LIN {X 0.032,Y -299.569,Z 1828.357,A 0.000,B 0.000,C 90.000,E1 64.229} C_DIS
LIN {X -0.106,Y -287.457,Z 1828.340,A 0.000,B 0.000,C 90.000,E1 61.257} C_DIS
LIN {X -0.056,Y -278.078,Z 1828.327,A 0.000,B 0.000,C 90.000,E1 58.869} C_DIS
LIN {X 0.072,Y -268.639,Z 1828.313,A 0.000,B 0.000,C 90.000,E1 56.421} C_DIS
LIN {X 0.019,Y -260.469,Z 1828.302,A 0.000,B 0.000,C 90.000,E1 54.322} C_DIS
LIN {X -0.032,Y -252.251,Z 1828.290,A 0.000,B 0.000,C 90.000,E1 52.190} C_DIS
LIN {X -0.029,Y -249.462,Z 1828.286,A 0.000,B 0.000,C 90.000,E1 51.457} C_DIS
LIN {X -0.079,Y -249.453,Z 1828.286,A 0.000,B 0.000,C 90.000,E1 51.457} C_DIS
LIN {X 0.072,Y -254.487,Z 1828.280,A 0.000,B 0.000,C 90.000,E1 50.356} C_DIS
LIN {X -0.079,Y -255.818,Z 1828.276,A 0.000,B 0.000,C 90.000,E1 49.666} C_DIS
LIN {X -0.023,Y -255.690,Z 1828.272,A 0.000,B 0.000,C 90.000,E1 48.933} C_DIS
LIN {X -0.153,Y -255.059,Z 1828.268,A 0.000,B 0.000,C 90.000,E1 48.243} C_DIS
LIN {X 0.076,Y -254.151,Z 1828.264,A 0.000,B 0.000,C 90.000,E1 47.472} C_DIS
LIN {X -0.026,Y -251.829,Z 1828.256,A 0.000,B 0.000,C 90.000,E1 46.053} C_DIS
LIN {X 0.022,Y -249.143,Z 1828.248,A 0.000,B 0.000,C 90.000,E1 44.595} C_DIS
LIN {X 0.039,Y -244.690,Z 1828.236,A 0.000,B 0.000,C 90.000,E1 42.405} C_DIS
LIN {X -0.033,Y -239.918,Z 1828.223,A 0.000,B 0.000,C 90.000,E1 40.216} C_DIS
LIN {X -0.009,Y -233.391,Z 1828.207,A 0.000,B 0.000,C 90.000,E1 37.237} C_DIS
LIN {X 0.086,Y -226.660,Z 1828.190,A 0.000,B 0.000,C 90.000,E1 34.199} C_DIS
LIN {X 0.024,Y -221.773,Z 1828.177,A 0.000,B 0.000,C 90.000,E1 31.926} C_DIS
LIN {X 0.052,Y -213.666,Z 1828.156,A 0.000,B 0.000,C 90.000,E1 28.052} C_DIS
LIN {X 0.010,Y -206.205,Z 1828.134,A 0.000,B 0.000,C 90.000,E1 24.131} C_DIS
LIN {X 0.086,Y -200.971,Z 1828.116,A 0.000,B 0.000,C 90.000,E1 20.918} C_DIS
LIN {X -0.033,Y -195.411,Z 1828.094,A 0.000,B 0.000,C 90.000,E1 16.913} C_DIS
LIN {X -0.035,Y -191.019,Z 1828.071,A 0.000,B 0.000,C 90.000,E1 12.827} C_DIS
LIN {X 0.032,Y -187.518,Z 1828.048,A 0.000,B 0.000,C 90.000,E1 8.681} C_DIS
LIN {X -0.001,Y -184.293,Z 1828.016,A 0.000,B 0.000,C 90.000,E1 2.865} C_DIS
LIN {X 0.059,Y -182.919,Z 1827.979,A 0.000,B 0.000,C 90.000,E1 356.159} C_DIS
LIN {X -0.023,Y -183.519,Z 1827.937,A 0.000,B 0.000,C 90.000,E1 348.634} C_DIS
LIN {X -0.034,Y -184.958,Z 1827.909,A 0.000,B 0.000,C 90.000,E1 343.614} C_DIS
LIN {X 0.018,Y -187.227,Z 1827.881,A 0.000,B 0.000,C 90.000,E1 338.592} C_DIS
LIN {X -0.063,Y -190.361,Z 1827.853,A 0.000,B 0.000,C 90.000,E1 333.640} C_DIS
LIN {X 0.062,Y -194.276,Z 1827.826,A 0.000,B 0.000,C 90.000,E1 328.663} C_DIS
LIN {X -0.035,Y -198.125,Z 1827.803,A 0.000,B 0.000,C 90.000,E1 324.609} C_DIS
LIN {X -0.033,Y -202.723,Z 1827.781,A 0.000,B 0.000,C 90.000,E1 320.561} C_DIS
LIN {X 0.128,Y -207.396,Z 1827.763,A 0.000,B 0.000,C 90.000,E1 317.310} C_DIS
LIN {X 0.009,Y -211.919,Z 1827.750,A 0.000,B 0.000,C 90.000,E1 314.960} C_DIS
LIN {X -0.077,Y -216.582,Z 1827.739,A 0.000,B 0.000,C 90.000,E1 313.014} C_DIS
LIN {X 0.005,Y -221.156,Z 1827.730,A 0.000,B 0.000,C 90.000,E1 311.434} C_DIS
LIN {X 0.022,Y -226.545,Z 1827.722,A 0.000,B 0.000,C 90.000,E1 309.886} C_DIS
LIN {X -0.066,Y -232.712,Z 1827.713,A 0.000,B 0.000,C 90.000,E1 308.382} C_DIS
LIN {X 0.102,Y -243.179,Z 1827.701,A 0.000,B 0.000,C 90.000,E1 306.091} C_DIS
LIN {X -0.019,Y -252.825,Z 1827.690,A 0.000,B 0.000,C 90.000,E1 304.278} C_DIS
LIN {X -0.093,Y -265.541,Z 1827.678,A 0.000,B 0.000,C 90.000,E1 302.133} C_DIS
LIN {X -0.090,Y -284.139,Z 1827.663,A 0.000,B 0.000,C 90.000,E1 299.333} C_DIS
LIN {X 0.121,Y -298.703,Z 1827.652,A 0.000,B 0.000,C 90.000,E1 297.257} C_DIS
LIN {X -0.090,Y -311.079,Z 1827.642,A 0.000,B 0.000,C 90.000,E1 295.643} C_DIS
LIN {X -0.108,Y -323.475,Z 1827.633,A 0.000,B 0.000,C 90.000,E1 294.027} C_DIS
LIN {X 0.094,Y -335.710,Z 1827.625,A 0.000,B 0.000,C 90.000,E1 292.408} C_DIS
LIN {X 0.045,Y -345.213,Z 1827.618,A 0.000,B 0.000,C 90.000,E1 291.173} C_DIS
LIN {X 0.112,Y -354.151,Z 1827.611,A 0.000,B 0.000,C 90.000,E1 289.939} C_DIS
LIN {X 0.111,Y -360.270,Z 1827.606,A 0.000,B 0.000,C 90.000,E1 289.033} C_DIS
LIN {X -0.171,Y -365.811,Z 1827.601,A 0.000,B 0.000,C 90.000,E1 288.181} C_DIS
LIN {X -0.063,Y -370.611,Z 1827.596,A 0.000,B 0.000,C 90.000,E1 287.275} C_DIS
LIN {X -0.011,Y -374.520,Z 1827.591,A 0.000,B 0.000,C 90.000,E1 286.386} C_DIS
LIN {X 0.180,Y -377.576,Z 1827.586,A 0.000,B 0.000,C 90.000,E1 285.481} C_DIS
LIN {X -0.181,Y -379.206,Z 1827.583,A 0.000,B 0.000,C 90.000,E1 284.954} C_DIS
LIN {X -0.066,Y -380.464,Z 1827.580,A 0.000,B 0.000,C 90.000,E1 284.356} C_DIS
LIN {X -0.035,Y -381.302,Z 1827.577,A 0.000,B 0.000,C 90.000,E1 283.772} C_DIS
LIN {X 0.094,Y -381.711,Z 1827.573,A 0.000,B 0.000,C 90.000,E1 283.175} C_DIS
LIN {X 0.140,Y -381.680,Z 1827.570,A 0.000,B 0.000,C 90.000,E1 282.591} C_DIS
LIN {X -0.183,Y -381.269,Z 1827.567,A 0.000,B 0.000,C 90.000,E1 282.063} C_DIS
LIN {X -0.132,Y -380.387,Z 1827.564,A 0.000,B 0.000,C 90.000,E1 281.478} C_DIS
LIN {X -0.084,Y -379.051,Z 1827.560,A 0.000,B 0.000,C 90.000,E1 280.894} C_DIS
LIN {X -0.042,Y -377.252,Z 1827.557,A 0.000,B 0.000,C 90.000,E1 280.310} C_DIS
LIN {X -0.060,Y -373.979,Z 1827.552,A 0.000,B 0.000,C 90.000,E1 279.443} C_DIS
LIN {X -0.118,Y -367.706,Z 1827.544,A 0.000,B 0.000,C 90.000,E1 277.992} C_DIS
LIN {X 0.139,Y -363.441,Z 1827.539,A 0.000,B 0.000,C 90.000,E1 277.068} C_DIS
LIN {X 0.076,Y -360.186,Z 1827.536,A 0.000,B 0.000,C 90.000,E1 276.486} C_DIS
LIN {X -0.130,Y -354.419,Z 1827.531,A 0.000,B 0.000,C 90.000,E1 275.625} C_DIS
LIN {X 0.069,Y -349.826,Z 1827.528,A 0.000,B 0.000,C 90.000,E1 274.992} C_DIS
LIN {X -0.106,Y -344.534,Z 1827.524,A 0.000,B 0.000,C 90.000,E1 274.416} C_DIS
LIN {X 0.153,Y -338.687,Z 1827.521,A 0.000,B 0.000,C 90.000,E1 273.784} C_DIS
LIN {X 0.006,Y -332.711,Z 1827.518,A 0.000,B 0.000,C 90.000,E1 273.269} C_DIS
LIN {X 0.134,Y -326.424,Z 1827.515,A 0.000,B 0.000,C 90.000,E1 272.751} C_DIS
LIN {X -0.129,Y -319.978,Z 1827.513,A 0.000,B 0.000,C 90.000,E1 272.350} C_DIS
LIN {X -0.138,Y -313.290,Z 1827.511,A 0.000,B 0.000,C 90.000,E1 271.949} C_DIS
LIN {X 0.132,Y -306.164,Z 1827.509,A 0.000,B 0.000,C 90.000,E1 271.547} C_DIS
LIN {X 0.043,Y -298.467,Z 1827.507,A 0.000,B 0.000,C 90.000,E1 271.260} C_DIS
LIN {X 0.041,Y -291.054,Z 1827.506,A 0.000,B 0.000,C 90.000,E1 271.031} C_DIS
LIN {X 0.116,Y -279.908,Z 1827.504,A 0.000,B 0.000,C 90.000,E1 270.745} C_DIS
LIN {X -0.065,Y -250.463,Z 1827.501,A 0.000,B 0.000,C 90.000,E1 270.229} C_DIS
LIN {X -0.110,Y -240.845,Z 1827.500,A 0.000,B 0.000,C 90.000,E1 270.115} C_DIS
LIN {X -0.045,Y -234.411,Z 1827.500,A 0.000,B 0.000,C 90.000,E1 270.057} C_DIS
LIN {X -0.062,Y -181.566,Z 1827.500,A 0.000,B 0.000,C 90.000,E1 270.057} C_DIS
LIN {X 0.021,Y -180.907,Z 1827.475,A 0.000,B 0.000,C 90.000,E1 265.469} C_DIS
LIN {X 0.079,Y -180.739,Z 1827.470,A 0.000,B 0.000,C 90.000,E1 264.609} C_DIS
LIN {X 0.000,Y -178.830,Z 1827.442,A 0.000,B 0.000,C 90.000,E1 259.567} C_DIS
LIN {X 0.033,Y -175.874,Z 1827.414,A 0.000,B 0.000,C 90.000,E1 254.464} C_DIS
LIN {X -0.090,Y -173.848,Z 1827.400,A 0.000,B 0.000,C 90.000,E1 251.945} C_DIS
LIN {X 0.064,Y -171.516,Z 1827.380,A 0.000,B 0.000,C 90.000,E1 248.465} C_DIS
LIN {X 0.049,Y -167.743,Z 1827.356,A 0.000,B 0.000,C 90.000,E1 244.152} C_DIS
LIN {X 0.065,Y -166.444,Z 1827.347,A 0.000,B 0.000,C 90.000,E1 242.410} C_DIS
LIN {X -0.021,Y -163.161,Z 1827.327,A 0.000,B 0.000,C 90.000,E1 238.948} C_DIS
LIN {X 0.028,Y -161.119,Z 1827.313,A 0.000,B 0.000,C 90.000,E1 236.294} C_DIS
LIN {X -0.069,Y -157.143,Z 1827.288,A 0.000,B 0.000,C 90.000,E1 231.904} C_DIS
LIN {X -0.046,Y -155.876,Z 1827.278,A 0.000,B 0.000,C 90.000,E1 230.114} C_DIS
LIN {X -0.087,Y -152.125,Z 1827.253,A 0.000,B 0.000,C 90.000,E1 225.648} C_DIS
LIN {X -0.067,Y -150.375,Z 1827.238,A 0.000,B 0.000,C 90.000,E1 222.933} C_DIS
LIN {X -0.042,Y -147.109,Z 1827.213,A 0.000,B 0.000,C 90.000,E1 218.382} C_DIS
LIN {X 0.068,Y -145.676,Z 1827.198,A 0.000,B 0.000,C 90.000,E1 215.598} C_DIS
LIN {X -0.052,Y -143.058,Z 1827.172,A 0.000,B 0.000,C 90.000,E1 211.052} C_DIS
LIN {X 0.006,Y -141.680,Z 1827.152,A 0.000,B 0.000,C 90.000,E1 207.334} C_DIS
LIN {X -0.016,Y -139.457,Z 1827.116,A 0.000,B 0.000,C 90.000,E1 200.844} C_DIS
LIN {X 0.035,Y -139.190,Z 1827.105,A 0.000,B 0.000,C 90.000,E1 198.960} C_DIS
LIN {X 0.058,Y -138.324,Z 1827.054,A 0.000,B 0.000,C 90.000,E1 189.613} C_DIS
LIN {X 0.066,Y -139.456,Z 1827.007,A 0.000,B 0.000,C 90.000,E1 181.203} C_DIS
LIN {X 0.007,Y -141.006,Z 1826.976,A 0.000,B 0.000,C 90.000,E1 175.641} C_DIS
LIN {X -0.044,Y -142.760,Z 1826.955,A 0.000,B 0.000,C 90.000,E1 171.951} C_DIS
LIN {X 0.053,Y -145.165,Z 1826.930,A 0.000,B 0.000,C 90.000,E1 167.297} C_DIS
LIN {X 0.045,Y -147.787,Z 1826.909,A 0.000,B 0.000,C 90.000,E1 163.630} C_DIS
LIN {X -0.018,Y -150.468,Z 1826.889,A 0.000,B 0.000,C 90.000,E1 160.007} C_DIS
LIN {X 0.056,Y -153.921,Z 1826.869,A 0.000,B 0.000,C 90.000,E1 156.357} C_DIS
LIN {X -0.020,Y -157.331,Z 1826.849,A 0.000,B 0.000,C 90.000,E1 152.794} C_DIS
LIN {X 0.065,Y -161.522,Z 1826.829,A 0.000,B 0.000,C 90.000,E1 149.203} C_DIS
LIN {X 0.078,Y -165.721,Z 1826.809,A 0.000,B 0.000,C 90.000,E1 145.674} C_DIS
LIN {X 0.066,Y -170.669,Z 1826.790,A 0.000,B 0.000,C 90.000,E1 142.190} C_DIS
LIN {X -0.021,Y -175.544,Z 1826.771,A 0.000,B 0.000,C 90.000,E1 138.771} C_DIS
LIN {X 0.099,Y -181.163,Z 1826.752,A 0.000,B 0.000,C 90.000,E1 135.324} C_DIS
LIN {X -0.031,Y -186.618,Z 1826.733,A 0.000,B 0.000,C 90.000,E1 132.000} C_DIS
LIN {X 0.039,Y -191.227,Z 1826.719,A 0.000,B 0.000,C 90.000,E1 129.483} C_DIS
LIN {X -0.039,Y -197.042,Z 1826.701,A 0.000,B 0.000,C 90.000,E1 126.217} C_DIS
LIN {X -0.121,Y -200.314,Z 1826.692,A 0.000,B 0.000,C 90.000,E1 124.612} C_DIS
LIN {X 0.050,Y -207.804,Z 1826.670,A 0.000,B 0.000,C 90.000,E1 120.541} C_DIS
LIN {X 0.057,Y -210.971,Z 1826.661,A 0.000,B 0.000,C 90.000,E1 118.949} C_DIS
LIN {X 0.072,Y -216.849,Z 1826.643,A 0.000,B 0.000,C 90.000,E1 115.796} C_DIS
LIN {X 0.026,Y -218.465,Z 1826.639,A 0.000,B 0.000,C 90.000,E1 115.027} C_DIS
LIN {X 0.067,Y -221.183,Z 1826.630,A 0.000,B 0.000,C 90.000,E1 113.462} C_DIS
LIN {X -0.050,Y -224.036,Z 1826.622,A 0.000,B 0.000,C 90.000,E1 111.897} C_DIS
LIN {X -0.098,Y -283.686,Z 1826.622,A 0.000,B 0.000,C 90.000,E1 111.897} C_DIS
LIN {X 0.024,Y -285.203,Z 1826.621,A 0.000,B 0.000,C 90.000,E1 111.844} C_DIS
LIN {X 0.074,Y -288.957,Z 1826.620,A 0.000,B 0.000,C 90.000,E1 111.663} C_DIS
LIN {X -0.144,Y -291.142,Z 1826.620,A 0.000,B 0.000,C 90.000,E1 111.535} C_DIS
LIN {X 0.064,Y -294.171,Z 1826.618,A 0.000,B 0.000,C 90.000,E1 111.153} C_DIS
LIN {X 0.041,Y -296.176,Z 1826.616,A 0.000,B 0.000,C 90.000,E1 110.844} C_DIS
LIN {X 0.051,Y -309.270,Z 1826.603,A 0.000,B 0.000,C 90.000,E1 108.544} C_DIS
LIN {X 0.157,Y -323.836,Z 1826.590,A 0.000,B 0.000,C 90.000,E1 106.260} C_DIS
LIN {X -0.113,Y -337.506,Z 1826.580,A 0.000,B 0.000,C 90.000,E1 104.411} C_DIS
LIN {X 0.033,Y -352.360,Z 1826.570,A 0.000,B 0.000,C 90.000,E1 102.535} C_DIS
LIN {X 0.042,Y -370.762,Z 1826.558,A 0.000,B 0.000,C 90.000,E1 100.489} C_DIS
LIN {X 0.113,Y -389.583,Z 1826.548,A 0.000,B 0.000,C 90.000,E1 98.624} C_DIS
LIN {X 0.008,Y -408.823,Z 1826.539,A 0.000,B 0.000,C 90.000,E1 96.947} C_DIS
LIN {X -0.185,Y -431.190,Z 1826.529,A 0.000,B 0.000,C 90.000,E1 95.220} C_DIS
LIN {X -0.025,Y -439.544,Z 1826.526,A 0.000,B 0.000,C 90.000,E1 94.588} C_DIS
LIN {X 0.191,Y -441.622,Z 1826.524,A 0.000,B 0.000,C 90.000,E1 94.359} C_DIS
LIN {X 0.043,Y -443.572,Z 1826.523,A 0.000,B 0.000,C 90.000,E1 94.131} C_DIS
LIN {X -0.076,Y -445.062,Z 1826.522,A 0.000,B 0.000,C 90.000,E1 93.898} C_DIS
LIN {X 0.104,Y -446.265,Z 1826.520,A 0.000,B 0.000,C 90.000,E1 93.612} C_DIS
LIN {X -0.161,Y -447.151,Z 1826.519,A 0.000,B 0.000,C 90.000,E1 93.383} C_DIS
LIN {X -0.205,Y -448.124,Z 1826.516,A 0.000,B 0.000,C 90.000,E1 92.865} C_DIS
LIN {X 0.183,Y -448.151,Z 1826.513,A 0.000,B 0.000,C 90.000,E1 92.293} C_DIS
LIN {X 0.144,Y -447.239,Z 1826.510,A 0.000,B 0.000,C 90.000,E1 91.776} C_DIS
LIN {X 0.091,Y -445.244,Z 1826.507,A 0.000,B 0.000,C 90.000,E1 91.260} C_DIS
LIN {X -0.041,Y -438.759,Z 1826.501,A 0.000,B 0.000,C 90.000,E1 90.229} C_DIS
LIN {X 0.192,Y -427.223,Z 1826.491,A 0.000,B 0.000,C 90.000,E1 88.339} C_DIS
LIN {X -0.201,Y -415.449,Z 1826.480,A 0.000,B 0.000,C 90.000,E1 86.502} C_DIS
LIN {X 0.029,Y -403.593,Z 1826.470,A 0.000,B 0.000,C 90.000,E1 84.546} C_DIS
LIN {X 0.006,Y -391.662,Z 1826.459,A 0.000,B 0.000,C 90.000,E1 82.591} C_DIS
LIN {X -0.174,Y -379.704,Z 1826.448,A 0.000,B 0.000,C 90.000,E1 80.622} C_DIS
LIN {X -0.113,Y -364.559,Z 1826.433,A 0.000,B 0.000,C 90.000,E1 77.993} C_DIS
LIN {X 0.006,Y -347.149,Z 1826.415,A 0.000,B 0.000,C 90.000,E1 74.685} C_DIS
LIN {X -0.011,Y -335.109,Z 1826.401,A 0.000,B 0.000,C 90.000,E1 72.236} C_DIS
LIN {X -0.116,Y -323.322,Z 1826.387,A 0.000,B 0.000,C 90.000,E1 69.752} C_DIS
LIN {X -0.027,Y -309.201,Z 1826.370,A 0.000,B 0.000,C 90.000,E1 66.538} C_DIS
LIN {X -0.176,Y -299.597,Z 1826.357,A 0.000,B 0.000,C 90.000,E1 64.280} C_DIS
LIN {X -0.044,Y -287.482,Z 1826.340,A 0.000,B 0.000,C 90.000,E1 61.257} C_DIS
LIN {X 0.004,Y -278.105,Z 1826.327,A 0.000,B 0.000,C 90.000,E1 58.869} C_DIS
LIN {X 0.130,Y -268.669,Z 1826.314,A 0.000,B 0.000,C 90.000,E1 56.421} C_DIS
LIN {X 0.077,Y -260.499,Z 1826.302,A 0.000,B 0.000,C 90.000,E1 54.322} C_DIS
LIN {X 0.062,Y -256.702,Z 1826.296,A 0.000,B 0.000,C 90.000,E1 53.336} C_DIS
LIN {X 0.012,Y -256.683,Z 1826.296,A 0.000,B 0.000,C 90.000,E1 53.336} C_DIS
LIN {X 0.030,Y -261.851,Z 1826.290,A 0.000,B 0.000,C 90.000,E1 52.190} C_DIS
LIN {X 0.074,Y -262.675,Z 1826.288,A 0.000,B 0.000,C 90.000,E1 51.823} C_DIS
LIN {X 0.015,Y -262.863,Z 1826.284,A 0.000,B 0.000,C 90.000,E1 51.126} C_DIS
LIN {X -0.079,Y -262.317,Z 1826.280,A 0.000,B 0.000,C 90.000,E1 50.436} C_DIS
LIN {X 0.032,Y -261.416,Z 1826.276,A 0.000,B 0.000,C 90.000,E1 49.703} C_DIS
LIN {X -0.158,Y -259.054,Z 1826.268,A 0.000,B 0.000,C 90.000,E1 48.324} C_DIS
LIN {X -0.009,Y -256.276,Z 1826.260,A 0.000,B 0.000,C 90.000,E1 46.863} C_DIS
LIN {X 0.133,Y -251.648,Z 1826.248,A 0.000,B 0.000,C 90.000,E1 44.676} C_DIS
LIN {X 0.012,Y -246.729,Z 1826.236,A 0.000,B 0.000,C 90.000,E1 42.528} C_DIS
LIN {X 0.002,Y -241.617,Z 1826.224,A 0.000,B 0.000,C 90.000,E1 40.334} C_DIS
LIN {X 0.032,Y -234.705,Z 1826.208,A 0.000,B 0.000,C 90.000,E1 37.363} C_DIS
LIN {X 0.025,Y -227.628,Z 1826.191,A 0.000,B 0.000,C 90.000,E1 34.358} C_DIS
LIN {X -0.014,Y -222.517,Z 1826.178,A 0.000,B 0.000,C 90.000,E1 32.084} C_DIS
LIN {X -0.042,Y -214.038,Z 1826.157,A 0.000,B 0.000,C 90.000,E1 28.231} C_DIS
LIN {X 0.026,Y -206.204,Z 1826.135,A 0.000,B 0.000,C 90.000,E1 24.283} C_DIS
LIN {X -0.002,Y -200.772,Z 1826.117,A 0.000,B 0.000,C 90.000,E1 21.099} C_DIS
LIN {X 0.062,Y -195.153,Z 1826.095,A 0.000,B 0.000,C 90.000,E1 17.040} C_DIS
LIN {X 0.056,Y -190.746,Z 1826.072,A 0.000,B 0.000,C 90.000,E1 12.952} C_DIS
LIN {X -0.064,Y -187.228,Z 1826.049,A 0.000,B 0.000,C 90.000,E1 8.859} C_DIS
LIN {X -0.087,Y -183.950,Z 1826.017,A 0.000,B 0.000,C 90.000,E1 3.037} C_DIS
LIN {X 0.049,Y -182.523,Z 1825.979,A 0.000,B 0.000,C 90.000,E1 356.159} C_DIS
LIN {X -0.054,Y -183.146,Z 1825.937,A 0.000,B 0.000,C 90.000,E1 348.634} C_DIS
LIN {X 0.097,Y -184.598,Z 1825.909,A 0.000,B 0.000,C 90.000,E1 343.559} C_DIS
LIN {X -0.041,Y -186.900,Z 1825.881,A 0.000,B 0.000,C 90.000,E1 338.592} C_DIS
LIN {X 0.035,Y -190.071,Z 1825.853,A 0.000,B 0.000,C 90.000,E1 333.589} C_DIS
LIN {X -0.023,Y -194.016,Z 1825.826,A 0.000,B 0.000,C 90.000,E1 328.663} C_DIS
LIN {X 0.032,Y -197.887,Z 1825.803,A 0.000,B 0.000,C 90.000,E1 324.562} C_DIS
LIN {X 0.021,Y -202.562,Z 1825.781,A 0.000,B 0.000,C 90.000,E1 320.517} C_DIS
LIN {X 0.019,Y -207.333,Z 1825.763,A 0.000,B 0.000,C 90.000,E1 317.310} C_DIS
LIN {X 0.047,Y -211.950,Z 1825.750,A 0.000,B 0.000,C 90.000,E1 314.919} C_DIS
LIN {X -0.043,Y -216.696,Z 1825.739,A 0.000,B 0.000,C 90.000,E1 312.975} C_DIS
LIN {X 0.055,Y -221.326,Z 1825.730,A 0.000,B 0.000,C 90.000,E1 311.391} C_DIS
LIN {X 0.052,Y -226.748,Z 1825.721,A 0.000,B 0.000,C 90.000,E1 309.850} C_DIS
LIN {X 0.001,Y -232.962,Z 1825.713,A 0.000,B 0.000,C 90.000,E1 308.338} C_DIS
LIN {X -0.015,Y -243.483,Z 1825.700,A 0.000,B 0.000,C 90.000,E1 306.091} C_DIS
LIN {X 0.007,Y -253.163,Z 1825.690,A 0.000,B 0.000,C 90.000,E1 304.246} C_DIS
LIN {X 0.122,Y -263.710,Z 1825.680,A 0.000,B 0.000,C 90.000,E1 302.418} C_DIS
LIN {X -0.147,Y -282.183,Z 1825.665,A 0.000,B 0.000,C 90.000,E1 299.667} C_DIS
LIN {X 0.024,Y -296.726,Z 1825.653,A 0.000,B 0.000,C 90.000,E1 297.590} C_DIS
LIN {X 0.084,Y -311.609,Z 1825.642,A 0.000,B 0.000,C 90.000,E1 295.591} C_DIS
LIN {X -0.079,Y -324.054,Z 1825.633,A 0.000,B 0.000,C 90.000,E1 294.003} C_DIS
LIN {X -0.002,Y -336.339,Z 1825.625,A 0.000,B 0.000,C 90.000,E1 292.408} C_DIS
LIN {X 0.079,Y -345.855,Z 1825.618,A 0.000,B 0.000,C 90.000,E1 291.153} C_DIS
LIN {X -0.006,Y -352.657,Z 1825.612,A 0.000,B 0.000,C 90.000,E1 290.248} C_DIS
LIN {X 0.104,Y -358.959,Z 1825.607,A 0.000,B 0.000,C 90.000,E1 289.322} C_DIS
LIN {X 0.146,Y -364.726,Z 1825.602,A 0.000,B 0.000,C 90.000,E1 288.417} C_DIS
LIN {X 0.171,Y -368.168,Z 1825.599,A 0.000,B 0.000,C 90.000,E1 287.819} C_DIS
LIN {X -0.134,Y -371.253,Z 1825.596,A 0.000,B 0.000,C 90.000,E1 287.275} C_DIS
LIN {X -0.068,Y -373.930,Z 1825.593,A 0.000,B 0.000,C 90.000,E1 286.677} C_DIS
LIN {X 0.019,Y -376.221,Z 1825.589,A 0.000,B 0.000,C 90.000,E1 286.079} C_DIS
LIN {X 0.119,Y -378.160,Z 1825.586,A 0.000,B 0.000,C 90.000,E1 285.481} C_DIS
LIN {X 0.128,Y -379.776,Z 1825.583,A 0.000,B 0.000,C 90.000,E1 284.898} C_DIS
LIN {X -0.121,Y -381.028,Z 1825.580,A 0.000,B 0.000,C 90.000,E1 284.356} C_DIS
LIN {X -0.087,Y -381.860,Z 1825.576,A 0.000,B 0.000,C 90.000,E1 283.772} C_DIS
LIN {X 0.046,Y -382.226,Z 1825.573,A 0.000,B 0.000,C 90.000,E1 283.175} C_DIS
LIN {X 0.096,Y -382.215,Z 1825.570,A 0.000,B 0.000,C 90.000,E1 282.591} C_DIS
LIN {X 0.149,Y -381.750,Z 1825.567,A 0.000,B 0.000,C 90.000,E1 282.007} C_DIS
LIN {X -0.170,Y -380.851,Z 1825.564,A 0.000,B 0.000,C 90.000,E1 281.478} C_DIS
LIN {X -0.119,Y -379.489,Z 1825.560,A 0.000,B 0.000,C 90.000,E1 280.894} C_DIS
LIN {X -0.074,Y -377.763,Z 1825.557,A 0.000,B 0.000,C 90.000,E1 280.310} C_DIS
LIN {X -0.088,Y -374.470,Z 1825.552,A 0.000,B 0.000,C 90.000,E1 279.443} C_DIS
LIN {X -0.137,Y -368.145,Z 1825.544,A 0.000,B 0.000,C 90.000,E1 277.992} C_DIS
LIN {X 0.124,Y -363.786,Z 1825.539,A 0.000,B 0.000,C 90.000,E1 277.068} C_DIS
LIN {X -0.013,Y -358.692,Z 1825.534,A 0.000,B 0.000,C 90.000,E1 276.201} C_DIS
LIN {X -0.140,Y -354.694,Z 1825.531,A 0.000,B 0.000,C 90.000,E1 275.625} C_DIS
LIN {X 0.062,Y -350.026,Z 1825.528,A 0.000,B 0.000,C 90.000,E1 274.992} C_DIS
LIN {X -0.014,Y -344.864,Z 1825.525,A 0.000,B 0.000,C 90.000,E1 274.416} C_DIS
LIN {X -0.067,Y -339.090,Z 1825.521,A 0.000,B 0.000,C 90.000,E1 273.841} C_DIS
LIN {X 0.095,Y -333.057,Z 1825.518,A 0.000,B 0.000,C 90.000,E1 273.269} C_DIS
LIN {X -0.101,Y -326.828,Z 1825.516,A 0.000,B 0.000,C 90.000,E1 272.808} C_DIS
LIN {X -0.058,Y -320.291,Z 1825.513,A 0.000,B 0.000,C 90.000,E1 272.350} C_DIS
LIN {X -0.029,Y -313.795,Z 1825.511,A 0.000,B 0.000,C 90.000,E1 271.949} C_DIS
LIN {X -0.081,Y -306.654,Z 1825.509,A 0.000,B 0.000,C 90.000,E1 271.604} C_DIS
LIN {X -0.133,Y -299.165,Z 1825.507,A 0.000,B 0.000,C 90.000,E1 271.318} C_DIS
LIN {X 0.139,Y -291.851,Z 1825.506,A 0.000,B 0.000,C 90.000,E1 271.031} C_DIS
LIN {X -0.083,Y -280.769,Z 1825.504,A 0.000,B 0.000,C 90.000,E1 270.802} C_DIS
LIN {X 0.009,Y -251.290,Z 1825.501,A 0.000,B 0.000,C 90.000,E1 270.229} C_DIS
LIN {X -0.042,Y -241.853,Z 1825.501,A 0.000,B 0.000,C 90.000,E1 270.115} C_DIS
LIN {X -0.019,Y -233.753,Z 1825.500,A 0.000,B 0.000,C 90.000,E1 270.057} C_DIS
LIN {X -0.042,Y -181.567,Z 1825.500,A 0.000,B 0.000,C 90.000,E1 270.057} C_DIS
LIN {X 0.066,Y -180.907,Z 1825.475,A 0.000,B 0.000,C 90.000,E1 265.469} C_DIS
LIN {X -0.056,Y -180.746,Z 1825.470,A 0.000,B 0.000,C 90.000,E1 264.666} C_DIS
LIN {X 0.012,Y -178.837,Z 1825.442,A 0.000,B 0.000,C 90.000,E1 259.577} C_DIS
LIN {X -0.092,Y -175.881,Z 1825.414,A 0.000,B 0.000,C 90.000,E1 254.519} C_DIS
LIN {X 0.015,Y -174.544,Z 1825.404,A 0.000,B 0.000,C 90.000,E1 252.779} C_DIS
LIN {X -0.053,Y -171.528,Z 1825.381,A 0.000,B 0.000,C 90.000,E1 248.518} C_DIS
LIN {X -0.059,Y -167.753,Z 1825.357,A 0.000,B 0.000,C 90.000,E1 244.204} C_DIS
LIN {X 0.031,Y -166.458,Z 1825.347,A 0.000,B 0.000,C 90.000,E1 242.436} C_DIS
LIN {X 0.021,Y -163.173,Z 1825.328,A 0.000,B 0.000,C 90.000,E1 238.948} C_DIS
LIN {X 0.070,Y -161.133,Z 1825.313,A 0.000,B 0.000,C 90.000,E1 236.294} C_DIS
LIN {X -0.027,Y -157.154,Z 1825.288,A 0.000,B 0.000,C 90.000,E1 231.904} C_DIS
LIN {X -0.004,Y -155.887,Z 1825.278,A 0.000,B 0.000,C 90.000,E1 230.114} C_DIS
LIN {X -0.046,Y -152.137,Z 1825.254,A 0.000,B 0.000,C 90.000,E1 225.648} C_DIS
LIN {X -0.026,Y -150.386,Z 1825.238,A 0.000,B 0.000,C 90.000,E1 222.933} C_DIS
LIN {X -0.002,Y -147.117,Z 1825.213,A 0.000,B 0.000,C 90.000,E1 218.382} C_DIS
LIN {X -0.011,Y -145.683,Z 1825.198,A 0.000,B 0.000,C 90.000,E1 215.644} C_DIS
LIN {X -0.012,Y -143.065,Z 1825.172,A 0.000,B 0.000,C 90.000,E1 211.052} C_DIS
LIN {X 0.045,Y -141.687,Z 1825.152,A 0.000,B 0.000,C 90.000,E1 207.334} C_DIS
LIN {X -0.027,Y -139.460,Z 1825.116,A 0.000,B 0.000,C 90.000,E1 200.865} C_DIS
LIN {X 0.074,Y -139.193,Z 1825.105,A 0.000,B 0.000,C 90.000,E1 198.960} C_DIS
LIN {X -0.040,Y -138.324,Z 1825.054,A 0.000,B 0.000,C 90.000,E1 189.670} C_DIS
LIN {X -0.035,Y -139.453,Z 1825.007,A 0.000,B 0.000,C 90.000,E1 181.260} C_DIS
LIN {X 0.045,Y -140.999,Z 1824.976,A 0.000,B 0.000,C 90.000,E1 175.641} C_DIS
LIN {X -0.005,Y -142.754,Z 1824.955,A 0.000,B 0.000,C 90.000,E1 171.951} C_DIS
LIN {X -0.050,Y -145.156,Z 1824.930,A 0.000,B 0.000,C 90.000,E1 167.353} C_DIS
LIN {X -0.056,Y -147.778,Z 1824.909,A 0.000,B 0.000,C 90.000,E1 163.685} C_DIS
LIN {X 0.023,Y -150.455,Z 1824.889,A 0.000,B 0.000,C 90.000,E1 160.007} C_DIS
LIN {X -0.044,Y -153.905,Z 1824.869,A 0.000,B 0.000,C 90.000,E1 156.410} C_DIS
LIN {X 0.022,Y -157.315,Z 1824.849,A 0.000,B 0.000,C 90.000,E1 152.794} C_DIS
LIN {X -0.032,Y -161.502,Z 1824.829,A 0.000,B 0.000,C 90.000,E1 149.253} C_DIS
LIN {X -0.017,Y -165.702,Z 1824.810,A 0.000,B 0.000,C 90.000,E1 145.722} C_DIS
LIN {X 0.110,Y -170.646,Z 1824.790,A 0.000,B 0.000,C 90.000,E1 142.190} C_DIS
LIN {X 0.023,Y -175.522,Z 1824.771,A 0.000,B 0.000,C 90.000,E1 138.771} C_DIS
LIN {X 0.017,Y -181.142,Z 1824.752,A 0.000,B 0.000,C 90.000,E1 135.364} C_DIS
LIN {X 0.015,Y -186.593,Z 1824.733,A 0.000,B 0.000,C 90.000,E1 132.000} C_DIS
LIN {X 0.085,Y -191.204,Z 1824.719,A 0.000,B 0.000,C 90.000,E1 129.483} C_DIS
LIN {X 0.009,Y -197.015,Z 1824.701,A 0.000,B 0.000,C 90.000,E1 126.217} C_DIS
LIN {X -0.073,Y -200.285,Z 1824.692,A 0.000,B 0.000,C 90.000,E1 124.612} C_DIS
LIN {X -0.080,Y -207.776,Z 1824.670,A 0.000,B 0.000,C 90.000,E1 120.590} C_DIS
LIN {X 0.106,Y -210.948,Z 1824.661,A 0.000,B 0.000,C 90.000,E1 118.949} C_DIS
LIN {X -0.073,Y -216.822,Z 1824.643,A 0.000,B 0.000,C 90.000,E1 115.848} C_DIS
LIN {X 0.075,Y -218.437,Z 1824.639,A 0.000,B 0.000,C 90.000,E1 115.027} C_DIS
LIN {X -0.085,Y -221.160,Z 1824.630,A 0.000,B 0.000,C 90.000,E1 113.515} C_DIS
LIN {X -0.027,Y -224.024,Z 1824.622,A 0.000,B 0.000,C 90.000,E1 111.897} C_DIS
LIN {X -0.069,Y -283.207,Z 1824.622,A 0.000,B 0.000,C 90.000,E1 111.897} C_DIS
LIN {X 0.089,Y -284.723,Z 1824.621,A 0.000,B 0.000,C 90.000,E1 111.844} C_DIS
LIN {X -0.128,Y -288.773,Z 1824.620,A 0.000,B 0.000,C 90.000,E1 111.716} C_DIS
LIN {X -0.078,Y -291.007,Z 1824.620,A 0.000,B 0.000,C 90.000,E1 111.535} C_DIS
LIN {X 0.024,Y -294.077,Z 1824.618,A 0.000,B 0.000,C 90.000,E1 111.173} C_DIS
LIN {X 0.019,Y -296.084,Z 1824.616,A 0.000,B 0.000,C 90.000,E1 110.865} C_DIS
LIN {X 0.153,Y -309.155,Z 1824.603,A 0.000,B 0.000,C 90.000,E1 108.544} C_DIS
LIN {X -0.049,Y -323.709,Z 1824.591,A 0.000,B 0.000,C 90.000,E1 106.315} C_DIS
LIN {X -0.006,Y -337.368,Z 1824.580,A 0.000,B 0.000,C 90.000,E1 104.411} C_DIS
LIN {X 0.141,Y -352.210,Z 1824.570,A 0.000,B 0.000,C 90.000,E1 102.535} C_DIS
LIN {X 0.146,Y -370.606,Z 1824.558,A 0.000,B 0.000,C 90.000,E1 100.489} C_DIS
LIN {X 0.213,Y -389.424,Z 1824.548,A 0.000,B 0.000,C 90.000,E1 98.624} C_DIS
LIN {X 0.103,Y -408.661,Z 1824.539,A 0.000,B 0.000,C 90.000,E1 96.947} C_DIS
LIN {X -0.094,Y -431.025,Z 1824.529,A 0.000,B 0.000,C 90.000,E1 95.220} C_DIS
LIN {X 0.063,Y -439.402,Z 1824.526,A 0.000,B 0.000,C 90.000,E1 94.588} C_DIS
LIN {X -0.162,Y -441.511,Z 1824.524,A 0.000,B 0.000,C 90.000,E1 94.416} C_DIS
LIN {X 0.149,Y -443.470,Z 1824.523,A 0.000,B 0.000,C 90.000,E1 94.131} C_DIS
LIN {X 0.049,Y -444.968,Z 1824.522,A 0.000,B 0.000,C 90.000,E1 93.898} C_DIS
LIN {X -0.216,Y -446.191,Z 1824.520,A 0.000,B 0.000,C 90.000,E1 93.669} C_DIS
LIN {X -0.036,Y -447.094,Z 1824.519,A 0.000,B 0.000,C 90.000,E1 93.383} C_DIS
LIN {X -0.079,Y -448.096,Z 1824.516,A 0.000,B 0.000,C 90.000,E1 92.865} C_DIS
LIN {X -0.140,Y -448.149,Z 1824.513,A 0.000,B 0.000,C 90.000,E1 92.350} C_DIS
LIN {X -0.178,Y -447.266,Z 1824.510,A 0.000,B 0.000,C 90.000,E1 91.833} C_DIS
LIN {X 0.215,Y -445.306,Z 1824.507,A 0.000,B 0.000,C 90.000,E1 91.260} C_DIS
LIN {X -0.101,Y -440.496,Z 1824.503,A 0.000,B 0.000,C 90.000,E1 90.516} C_DIS
LIN {X 0.176,Y -428.964,Z 1824.492,A 0.000,B 0.000,C 90.000,E1 88.625} C_DIS
LIN {X -0.188,Y -417.204,Z 1824.482,A 0.000,B 0.000,C 90.000,E1 86.788} C_DIS
LIN {X -0.016,Y -407.075,Z 1824.473,A 0.000,B 0.000,C 90.000,E1 85.122} C_DIS
LIN {X 0.038,Y -395.163,Z 1824.462,A 0.000,B 0.000,C 90.000,E1 83.166} C_DIS
LIN {X -0.068,Y -383.207,Z 1824.451,A 0.000,B 0.000,C 90.000,E1 81.197} C_DIS
LIN {X 0.023,Y -369.613,Z 1824.438,A 0.000,B 0.000,C 90.000,E1 78.870} C_DIS
LIN {X 0.132,Y -351.845,Z 1824.420,A 0.000,B 0.000,C 90.000,E1 75.589} C_DIS
LIN {X 0.109,Y -338.160,Z 1824.405,A 0.000,B 0.000,C 90.000,E1 72.851} C_DIS
LIN {X 0.099,Y -327.784,Z 1824.393,A 0.000,B 0.000,C 90.000,E1 70.678} C_DIS
LIN {X -0.102,Y -313.419,Z 1824.375,A 0.000,B 0.000,C 90.000,E1 67.539} C_DIS
LIN {X 0.013,Y -302.403,Z 1824.361,A 0.000,B 0.000,C 90.000,E1 64.921} C_DIS
LIN {X -0.042,Y -290.191,Z 1824.344,A 0.000,B 0.000,C 90.000,E1 61.948} C_DIS
LIN {X -0.066,Y -280.836,Z 1824.331,A 0.000,B 0.000,C 90.000,E1 59.587} C_DIS
LIN {X -0.017,Y -271.430,Z 1824.318,A 0.000,B 0.000,C 90.000,E1 57.168} C_DIS
LIN {X -0.038,Y -263.914,Z 1824.307,A 0.000,B 0.000,C 90.000,E1 55.229} C_DIS
LIN {X 0.128,Y -263.915,Z 1824.307,A 0.000,B 0.000,C 90.000,E1 55.182} C_DIS
LIN {X 0.081,Y -269.153,Z 1824.300,A 0.000,B 0.000,C 90.000,E1 53.989} C_DIS
LIN {X 0.063,Y -270.130,Z 1824.296,A 0.000,B 0.000,C 90.000,E1 53.290} C_DIS
LIN {X 0.002,Y -269.793,Z 1824.292,A 0.000,B 0.000,C 90.000,E1 52.603} C_DIS
LIN {X -0.001,Y -268.969,Z 1824.288,A 0.000,B 0.000,C 90.000,E1 51.904} C_DIS
LIN {X 0.157,Y -267.876,Z 1824.284,A 0.000,B 0.000,C 90.000,E1 51.170} C_DIS
LIN {X -0.127,Y -265.185,Z 1824.277,A 0.000,B 0.000,C 90.000,E1 49.828} C_DIS
LIN {X 0.026,Y -260.528,Z 1824.265,A 0.000,B 0.000,C 90.000,E1 47.676} C_DIS
LIN {X -0.102,Y -255.486,Z 1824.253,A 0.000,B 0.000,C 90.000,E1 45.567} C_DIS
LIN {X 0.026,Y -250.266,Z 1824.241,A 0.000,B 0.000,C 90.000,E1 43.380} C_DIS
LIN {X -0.105,Y -244.870,Z 1824.229,A 0.000,B 0.000,C 90.000,E1 41.229} C_DIS
LIN {X 0.011,Y -237.582,Z 1824.213,A 0.000,B 0.000,C 90.000,E1 38.257} C_DIS
LIN {X 0.048,Y -232.108,Z 1824.200,A 0.000,B 0.000,C 90.000,E1 36.011} C_DIS
LIN {X 0.099,Y -223.071,Z 1824.179,A 0.000,B 0.000,C 90.000,E1 32.212} C_DIS
LIN {X 0.010,Y -215.940,Z 1824.162,A 0.000,B 0.000,C 90.000,E1 29.155} C_DIS
LIN {X 0.016,Y -209.224,Z 1824.145,A 0.000,B 0.000,C 90.000,E1 26.027} C_DIS
LIN {X 0.055,Y -203.189,Z 1824.127,A 0.000,B 0.000,C 90.000,E1 22.845} C_DIS
LIN {X 0.061,Y -198.188,Z 1824.109,A 0.000,B 0.000,C 90.000,E1 19.631} C_DIS
LIN {X 0.052,Y -193.941,Z 1824.091,A 0.000,B 0.000,C 90.000,E1 16.386} C_DIS
LIN {X 0.008,Y -189.666,Z 1824.068,A 0.000,B 0.000,C 90.000,E1 12.299} C_DIS
LIN {X 0.002,Y -186.357,Z 1824.045,A 0.000,B 0.000,C 90.000,E1 8.163} C_DIS
LIN {X -0.088,Y -183.292,Z 1824.013,A 0.000,B 0.000,C 90.000,E1 2.350} C_DIS
LIN {X -0.077,Y -182.068,Z 1823.974,A 0.000,B 0.000,C 90.000,E1 355.355} C_DIS
LIN {X 0.093,Y -182.763,Z 1823.937,A 0.000,B 0.000,C 90.000,E1 348.578} C_DIS
LIN {X 0.051,Y -184.230,Z 1823.909,A 0.000,B 0.000,C 90.000,E1 343.559} C_DIS
LIN {X 0.029,Y -187.035,Z 1823.876,A 0.000,B 0.000,C 90.000,E1 337.720} C_DIS
LIN {X 0.022,Y -190.385,Z 1823.849,A 0.000,B 0.000,C 90.000,E1 332.743} C_DIS
LIN {X 0.077,Y -194.510,Z 1823.821,A 0.000,B 0.000,C 90.000,E1 327.788} C_DIS
LIN {X 0.096,Y -198.543,Z 1823.798,A 0.000,B 0.000,C 90.000,E1 323.703} C_DIS
LIN {X -0.051,Y -203.547,Z 1823.776,A 0.000,B 0.000,C 90.000,E1 319.703} C_DIS
LIN {X -0.089,Y -207.293,Z 1823.763,A 0.000,B 0.000,C 90.000,E1 317.310} C_DIS
LIN {X -0.065,Y -211.994,Z 1823.750,A 0.000,B 0.000,C 90.000,E1 314.919} C_DIS
LIN {X 0.001,Y -216.821,Z 1823.739,A 0.000,B 0.000,C 90.000,E1 312.933} C_DIS
LIN {X -0.060,Y -221.499,Z 1823.730,A 0.000,B 0.000,C 90.000,E1 311.391} C_DIS
LIN {X -0.064,Y -226.964,Z 1823.721,A 0.000,B 0.000,C 90.000,E1 309.850} C_DIS
LIN {X 0.029,Y -233.212,Z 1823.713,A 0.000,B 0.000,C 90.000,E1 308.302} C_DIS
LIN {X 0.032,Y -241.931,Z 1823.702,A 0.000,B 0.000,C 90.000,E1 306.423} C_DIS
LIN {X -0.110,Y -251.498,Z 1823.692,A 0.000,B 0.000,C 90.000,E1 304.612} C_DIS
LIN {X 0.112,Y -261.921,Z 1823.682,A 0.000,B 0.000,C 90.000,E1 302.752} C_DIS
LIN {X 0.037,Y -280.230,Z 1823.666,A 0.000,B 0.000,C 90.000,E1 299.951} C_DIS
LIN {X 0.061,Y -294.763,Z 1823.655,A 0.000,B 0.000,C 90.000,E1 297.897} C_DIS
LIN {X -0.023,Y -312.139,Z 1823.642,A 0.000,B 0.000,C 90.000,E1 295.591} C_DIS
LIN {X 0.116,Y -324.656,Z 1823.633,A 0.000,B 0.000,C 90.000,E1 293.951} C_DIS
LIN {X 0.029,Y -336.969,Z 1823.624,A 0.000,B 0.000,C 90.000,E1 292.386} C_DIS
LIN {X -0.012,Y -346.498,Z 1823.618,A 0.000,B 0.000,C 90.000,E1 291.153} C_DIS
LIN {X -0.092,Y -353.322,Z 1823.612,A 0.000,B 0.000,C 90.000,E1 290.248} C_DIS
LIN {X 0.022,Y -359.619,Z 1823.607,A 0.000,B 0.000,C 90.000,E1 289.322} C_DIS
LIN {X 0.070,Y -365.395,Z 1823.602,A 0.000,B 0.000,C 90.000,E1 288.417} C_DIS
LIN {X 0.180,Y -370.401,Z 1823.597,A 0.000,B 0.000,C 90.000,E1 287.511} C_DIS
LIN {X -0.134,Y -374.500,Z 1823.593,A 0.000,B 0.000,C 90.000,E1 286.677} C_DIS
LIN {X -0.045,Y -376.828,Z 1823.589,A 0.000,B 0.000,C 90.000,E1 286.079} C_DIS
LIN {X 0.059,Y -378.772,Z 1823.586,A 0.000,B 0.000,C 90.000,E1 285.481} C_DIS
LIN {X 0.072,Y -380.353,Z 1823.583,A 0.000,B 0.000,C 90.000,E1 284.898} C_DIS
LIN {X 0.196,Y -381.559,Z 1823.580,A 0.000,B 0.000,C 90.000,E1 284.300} C_DIS
LIN {X -0.136,Y -382.404,Z 1823.576,A 0.000,B 0.000,C 90.000,E1 283.772} C_DIS
LIN {X -0.001,Y -382.751,Z 1823.573,A 0.000,B 0.000,C 90.000,E1 283.175} C_DIS
LIN {X 0.053,Y -382.712,Z 1823.570,A 0.000,B 0.000,C 90.000,E1 282.591} C_DIS
LIN {X 0.109,Y -382.240,Z 1823.567,A 0.000,B 0.000,C 90.000,E1 282.007} C_DIS
LIN {X 0.166,Y -381.323,Z 1823.564,A 0.000,B 0.000,C 90.000,E1 281.422} C_DIS
LIN {X -0.153,Y -379.936,Z 1823.560,A 0.000,B 0.000,C 90.000,E1 280.894} C_DIS
LIN {X -0.104,Y -378.249,Z 1823.557,A 0.000,B 0.000,C 90.000,E1 280.310} C_DIS
LIN {X -0.114,Y -374.957,Z 1823.552,A 0.000,B 0.000,C 90.000,E1 279.443} C_DIS
LIN {X -0.099,Y -369.947,Z 1823.546,A 0.000,B 0.000,C 90.000,E1 278.276} C_DIS
LIN {X 0.179,Y -365.719,Z 1823.541,A 0.000,B 0.000,C 90.000,E1 277.352} C_DIS
LIN {X 0.051,Y -360.822,Z 1823.536,A 0.000,B 0.000,C 90.000,E1 276.486} C_DIS
LIN {X -0.068,Y -357.026,Z 1823.533,A 0.000,B 0.000,C 90.000,E1 275.910} C_DIS
LIN {X 0.146,Y -352.694,Z 1823.529,A 0.000,B 0.000,C 90.000,E1 275.277} C_DIS
LIN {X -0.017,Y -347.677,Z 1823.526,A 0.000,B 0.000,C 90.000,E1 274.702} C_DIS
LIN {X -0.146,Y -342.091,Z 1823.523,A 0.000,B 0.000,C 90.000,E1 274.131} C_DIS
LIN {X -0.074,Y -336.208,Z 1823.520,A 0.000,B 0.000,C 90.000,E1 273.555} C_DIS
LIN {X -0.083,Y -330.038,Z 1823.517,A 0.000,B 0.000,C 90.000,E1 273.037} C_DIS
LIN {X -0.156,Y -323.702,Z 1823.514,A 0.000,B 0.000,C 90.000,E1 272.579} C_DIS
LIN {X 0.058,Y -317.179,Z 1823.512,A 0.000,B 0.000,C 90.000,E1 272.121} C_DIS
LIN {X -0.090,Y -310.404,Z 1823.510,A 0.000,B 0.000,C 90.000,E1 271.776} C_DIS
LIN {X 0.030,Y -303.134,Z 1823.508,A 0.000,B 0.000,C 90.000,E1 271.432} C_DIS
LIN {X 0.148,Y -295.786,Z 1823.506,A 0.000,B 0.000,C 90.000,E1 271.146} C_DIS
LIN {X -0.076,Y -288.248,Z 1823.505,A 0.000,B 0.000,C 90.000,E1 270.974} C_DIS
LIN {X 0.082,Y -276.819,Z 1823.504,A 0.000,B 0.000,C 90.000,E1 270.688} C_DIS
LIN {X 0.027,Y -251.365,Z 1823.501,A 0.000,B 0.000,C 90.000,E1 270.229} C_DIS
LIN {X -0.022,Y -241.811,Z 1823.501,A 0.000,B 0.000,C 90.000,E1 270.115} C_DIS
LIN {X 0.003,Y -232.894,Z 1823.500,A 0.000,B 0.000,C 90.000,E1 270.057} C_DIS
LIN {X -0.025,Y -181.568,Z 1823.500,A 0.000,B 0.000,C 90.000,E1 270.057} C_DIS
LIN {X 0.084,Y -180.907,Z 1823.475,A 0.000,B 0.000,C 90.000,E1 265.469} C_DIS
LIN {X -0.039,Y -180.748,Z 1823.470,A 0.000,B 0.000,C 90.000,E1 264.666} C_DIS
LIN {X 0.029,Y -178.840,Z 1823.442,A 0.000,B 0.000,C 90.000,E1 259.577} C_DIS
LIN {X -0.075,Y -175.883,Z 1823.414,A 0.000,B 0.000,C 90.000,E1 254.519} C_DIS
LIN {X 0.032,Y -174.548,Z 1823.404,A 0.000,B 0.000,C 90.000,E1 252.779} C_DIS
LIN {X -0.035,Y -171.533,Z 1823.381,A 0.000,B 0.000,C 90.000,E1 248.518} C_DIS
LIN {X -0.042,Y -167.758,Z 1823.357,A 0.000,B 0.000,C 90.000,E1 244.204} C_DIS
LIN {X -0.100,Y -166.463,Z 1823.347,A 0.000,B 0.000,C 90.000,E1 242.487} C_DIS
LIN {X 0.036,Y -163.178,Z 1823.328,A 0.000,B 0.000,C 90.000,E1 238.948} C_DIS
LIN {X -0.048,Y -161.138,Z 1823.313,A 0.000,B 0.000,C 90.000,E1 236.342} C_DIS
LIN {X -0.012,Y -157.158,Z 1823.288,A 0.000,B 0.000,C 90.000,E1 231.904} C_DIS
LIN {X 0.011,Y -155.891,Z 1823.278,A 0.000,B 0.000,C 90.000,E1 230.114} C_DIS
LIN {X -0.031,Y -152.140,Z 1823.254,A 0.000,B 0.000,C 90.000,E1 225.648} C_DIS
LIN {X -0.011,Y -150.390,Z 1823.239,A 0.000,B 0.000,C 90.000,E1 222.933} C_DIS
LIN {X 0.013,Y -147.121,Z 1823.213,A 0.000,B 0.000,C 90.000,E1 218.382} C_DIS
LIN {X 0.005,Y -145.686,Z 1823.198,A 0.000,B 0.000,C 90.000,E1 215.644} C_DIS
LIN {X 0.002,Y -143.068,Z 1823.172,A 0.000,B 0.000,C 90.000,E1 211.052} C_DIS
LIN {X -0.067,Y -141.689,Z 1823.152,A 0.000,B 0.000,C 90.000,E1 207.385} C_DIS
LIN {X -0.012,Y -139.461,Z 1823.116,A 0.000,B 0.000,C 90.000,E1 200.865} C_DIS
LIN {X -0.043,Y -139.194,Z 1823.106,A 0.000,B 0.000,C 90.000,E1 199.014} C_DIS
LIN {X -0.025,Y -138.325,Z 1823.054,A 0.000,B 0.000,C 90.000,E1 189.670} C_DIS
LIN {X -0.020,Y -139.451,Z 1823.007,A 0.000,B 0.000,C 90.000,E1 181.260} C_DIS
LIN {X 0.060,Y -140.997,Z 1822.976,A 0.000,B 0.000,C 90.000,E1 175.641} C_DIS
LIN {X 0.009,Y -142.751,Z 1822.955,A 0.000,B 0.000,C 90.000,E1 171.951} C_DIS
LIN {X -0.034,Y -145.151,Z 1822.930,A 0.000,B 0.000,C 90.000,E1 167.353} C_DIS
LIN {X -0.042,Y -147.774,Z 1822.909,A 0.000,B 0.000,C 90.000,E1 163.685} C_DIS
LIN {X 0.038,Y -150.450,Z 1822.889,A 0.000,B 0.000,C 90.000,E1 160.007} C_DIS
LIN {X -0.028,Y -153.898,Z 1822.869,A 0.000,B 0.000,C 90.000,E1 156.410} C_DIS
LIN {X 0.038,Y -157.309,Z 1822.849,A 0.000,B 0.000,C 90.000,E1 152.794} C_DIS
LIN {X -0.016,Y -161.495,Z 1822.829,A 0.000,B 0.000,C 90.000,E1 149.253} C_DIS
LIN {X 0.000,Y -165.694,Z 1822.810,A 0.000,B 0.000,C 90.000,E1 145.722} C_DIS
LIN {X -0.113,Y -170.638,Z 1822.790,A 0.000,B 0.000,C 90.000,E1 142.271} C_DIS
LIN {X 0.039,Y -175.513,Z 1822.771,A 0.000,B 0.000,C 90.000,E1 138.771} C_DIS
LIN {X -0.094,Y -181.134,Z 1822.752,A 0.000,B 0.000,C 90.000,E1 135.405} C_DIS
LIN {X 0.032,Y -186.584,Z 1822.733,A 0.000,B 0.000,C 90.000,E1 132.000} C_DIS
LIN {X -0.018,Y -191.196,Z 1822.719,A 0.000,B 0.000,C 90.000,E1 129.519} C_DIS
LIN {X 0.027,Y -197.005,Z 1822.701,A 0.000,B 0.000,C 90.000,E1 126.217} C_DIS
LIN {X -0.054,Y -200.275,Z 1822.692,A 0.000,B 0.000,C 90.000,E1 124.612} C_DIS
LIN {X -0.061,Y -207.766,Z 1822.670,A 0.000,B 0.000,C 90.000,E1 120.590} C_DIS
LIN {X -0.059,Y -210.939,Z 1822.661,A 0.000,B 0.000,C 90.000,E1 118.999} C_DIS
LIN {X -0.053,Y -216.811,Z 1822.644,A 0.000,B 0.000,C 90.000,E1 115.848} C_DIS
LIN {X 0.094,Y -218.427,Z 1822.639,A 0.000,B 0.000,C 90.000,E1 115.027} C_DIS
LIN {X -0.065,Y -221.153,Z 1822.630,A 0.000,B 0.000,C 90.000,E1 113.515} C_DIS
LIN {X -0.035,Y -224.028,Z 1822.622,A 0.000,B 0.000,C 90.000,E1 111.897} C_DIS
LIN {X -0.080,Y -283.639,Z 1822.622,A 0.000,B 0.000,C 90.000,E1 111.897} C_DIS
LIN {X -0.103,Y -288.712,Z 1822.620,A 0.000,B 0.000,C 90.000,E1 111.716} C_DIS
LIN {X -0.053,Y -290.961,Z 1822.620,A 0.000,B 0.000,C 90.000,E1 111.535} C_DIS
LIN {X 0.049,Y -294.042,Z 1822.618,A 0.000,B 0.000,C 90.000,E1 111.173} C_DIS
LIN {X 0.049,Y -296.049,Z 1822.616,A 0.000,B 0.000,C 90.000,E1 110.865} C_DIS
LIN {X -0.104,Y -309.114,Z 1822.603,A 0.000,B 0.000,C 90.000,E1 108.598} C_DIS
LIN {X -0.012,Y -323.663,Z 1822.591,A 0.000,B 0.000,C 90.000,E1 106.315} C_DIS
LIN {X 0.030,Y -337.318,Z 1822.580,A 0.000,B 0.000,C 90.000,E1 104.411} C_DIS
LIN {X -0.165,Y -352.156,Z 1822.570,A 0.000,B 0.000,C 90.000,E1 102.591} C_DIS
LIN {X -0.181,Y -370.550,Z 1822.558,A 0.000,B 0.000,C 90.000,E1 100.546} C_DIS
LIN {X -0.137,Y -389.368,Z 1822.548,A 0.000,B 0.000,C 90.000,E1 98.681} C_DIS
LIN {X 0.136,Y -408.603,Z 1822.539,A 0.000,B 0.000,C 90.000,E1 96.947} C_DIS
LIN {X -0.062,Y -430.966,Z 1822.529,A 0.000,B 0.000,C 90.000,E1 95.220} C_DIS
LIN {X 0.095,Y -439.348,Z 1822.526,A 0.000,B 0.000,C 90.000,E1 94.588} C_DIS
LIN {X -0.131,Y -441.469,Z 1822.524,A 0.000,B 0.000,C 90.000,E1 94.416} C_DIS
LIN {X 0.186,Y -443.429,Z 1822.523,A 0.000,B 0.000,C 90.000,E1 94.131} C_DIS
LIN {X 0.092,Y -444.929,Z 1822.522,A 0.000,B 0.000,C 90.000,E1 93.898} C_DIS
LIN {X -0.174,Y -446.158,Z 1822.520,A 0.000,B 0.000,C 90.000,E1 93.669} C_DIS
LIN {X 0.006,Y -447.068,Z 1822.519,A 0.000,B 0.000,C 90.000,E1 93.383} C_DIS
LIN {X -0.037,Y -448.078,Z 1822.516,A 0.000,B 0.000,C 90.000,E1 92.865} C_DIS
LIN {X -0.099,Y -448.140,Z 1822.513,A 0.000,B 0.000,C 90.000,E1 92.350} C_DIS
LIN {X -0.151,Y -447.264,Z 1822.510,A 0.000,B 0.000,C 90.000,E1 91.835} C_DIS
LIN {X -0.189,Y -445.316,Z 1822.507,A 0.000,B 0.000,C 90.000,E1 91.318} C_DIS
LIN {X -0.060,Y -440.512,Z 1822.503,A 0.000,B 0.000,C 90.000,E1 90.516} C_DIS
LIN {X -0.212,Y -428.979,Z 1822.493,A 0.000,B 0.000,C 90.000,E1 88.682} C_DIS
LIN {X -0.148,Y -417.219,Z 1822.482,A 0.000,B 0.000,C 90.000,E1 86.788} C_DIS
LIN {X 0.024,Y -407.089,Z 1822.473,A 0.000,B 0.000,C 90.000,E1 85.122} C_DIS
LIN {X 0.076,Y -395.178,Z 1822.462,A 0.000,B 0.000,C 90.000,E1 83.166} C_DIS
LIN {X -0.030,Y -383.224,Z 1822.451,A 0.000,B 0.000,C 90.000,E1 81.197} C_DIS
LIN {X 0.059,Y -369.627,Z 1822.438,A 0.000,B 0.000,C 90.000,E1 78.870} C_DIS
LIN {X -0.173,Y -351.856,Z 1822.420,A 0.000,B 0.000,C 90.000,E1 75.644} C_DIS
LIN {X -0.180,Y -338.168,Z 1822.405,A 0.000,B 0.000,C 90.000,E1 72.906} C_DIS
LIN {X 0.132,Y -327.790,Z 1822.393,A 0.000,B 0.000,C 90.000,E1 70.678} C_DIS
LIN {X -0.069,Y -313.424,Z 1822.375,A 0.000,B 0.000,C 90.000,E1 67.539} C_DIS
LIN {X 0.145,Y -303.783,Z 1822.363,A 0.000,B 0.000,C 90.000,E1 65.229} C_DIS
LIN {X -0.005,Y -292.842,Z 1822.348,A 0.000,B 0.000,C 90.000,E1 62.615} C_DIS
LIN {X 0.043,Y -284.862,Z 1822.337,A 0.000,B 0.000,C 90.000,E1 60.589} C_DIS
LIN {X 0.035,Y -275.477,Z 1822.323,A 0.000,B 0.000,C 90.000,E1 58.201} C_DIS
LIN {X -0.025,Y -271.100,Z 1822.317,A 0.000,B 0.000,C 90.000,E1 57.089} C_DIS
LIN {X 0.151,Y -271.076,Z 1822.317,A 0.000,B 0.000,C 90.000,E1 57.041} C_DIS
LIN {X -0.111,Y -276.511,Z 1822.310,A 0.000,B 0.000,C 90.000,E1 55.801} C_DIS
LIN {X -0.022,Y -277.310,Z 1822.308,A 0.000,B 0.000,C 90.000,E1 55.435} C_DIS
LIN {X -0.139,Y -277.409,Z 1822.304,A 0.000,B 0.000,C 90.000,E1 54.769} C_DIS
LIN {X -0.095,Y -276.738,Z 1822.300,A 0.000,B 0.000,C 90.000,E1 54.069} C_DIS
LIN {X 0.114,Y -275.692,Z 1822.296,A 0.000,B 0.000,C 90.000,E1 53.336} C_DIS
LIN {X -0.034,Y -272.957,Z 1822.289,A 0.000,B 0.000,C 90.000,E1 51.984} C_DIS
LIN {X -0.048,Y -269.811,Z 1822.281,A 0.000,B 0.000,C 90.000,E1 50.598} C_DIS
LIN {X 0.012,Y -264.619,Z 1822.269,A 0.000,B 0.000,C 90.000,E1 48.485} C_DIS
LIN {X -0.046,Y -259.216,Z 1822.258,A 0.000,B 0.000,C 90.000,E1 46.377} C_DIS
LIN {X 0.153,Y -253.660,Z 1822.246,A 0.000,B 0.000,C 90.000,E1 44.190} C_DIS
LIN {X -0.101,Y -248.030,Z 1822.234,A 0.000,B 0.000,C 90.000,E1 42.081} C_DIS
LIN {X 0.074,Y -242.321,Z 1822.221,A 0.000,B 0.000,C 90.000,E1 39.850} C_DIS
LIN {X -0.037,Y -234.734,Z 1822.205,A 0.000,B 0.000,C 90.000,E1 36.916} C_DIS
LIN {X -0.048,Y -227.070,Z 1822.188,A 0.000,B 0.000,C 90.000,E1 33.913} C_DIS
LIN {X 0.084,Y -221.533,Z 1822.176,A 0.000,B 0.000,C 90.000,E1 31.592} C_DIS
LIN {X -0.049,Y -214.178,Z 1822.158,A 0.000,B 0.000,C 90.000,E1 28.537} C_DIS
LIN {X -0.091,Y -207.509,Z 1822.141,A 0.000,B 0.000,C 90.000,E1 25.412} C_DIS
LIN {X -0.078,Y -203.007,Z 1822.128,A 0.000,B 0.000,C 90.000,E1 23.025} C_DIS
LIN {X -0.074,Y -197.951,Z 1822.110,A 0.000,B 0.000,C 90.000,E1 19.812} C_DIS
LIN {X -0.032,Y -193.673,Z 1822.092,A 0.000,B 0.000,C 90.000,E1 16.551} C_DIS
LIN {X 0.093,Y -189.349,Z 1822.069,A 0.000,B 0.000,C 90.000,E1 12.411} C_DIS
LIN {X 0.071,Y -186.034,Z 1822.046,A 0.000,B 0.000,C 90.000,E1 8.276} C_DIS
LIN {X -0.038,Y -182.945,Z 1822.014,A 0.000,B 0.000,C 90.000,E1 2.465} C_DIS
LIN {X -0.089,Y -181.684,Z 1821.974,A 0.000,B 0.000,C 90.000,E1 355.355} C_DIS
LIN {X 0.062,Y -182.365,Z 1821.937,A 0.000,B 0.000,C 90.000,E1 348.578} C_DIS
LIN {X 0.004,Y -183.856,Z 1821.909,A 0.000,B 0.000,C 90.000,E1 343.559} C_DIS
LIN {X -0.035,Y -186.710,Z 1821.876,A 0.000,B 0.000,C 90.000,E1 337.720} C_DIS
LIN {X -0.054,Y -190.094,Z 1821.849,A 0.000,B 0.000,C 90.000,E1 332.743} C_DIS
LIN {X -0.011,Y -194.261,Z 1821.821,A 0.000,B 0.000,C 90.000,E1 327.788} C_DIS
LIN {X -0.001,Y -198.330,Z 1821.798,A 0.000,B 0.000,C 90.000,E1 323.703} C_DIS
LIN {X -0.026,Y -203.446,Z 1821.776,A 0.000,B 0.000,C 90.000,E1 319.666} C_DIS
LIN {X 0.093,Y -207.284,Z 1821.763,A 0.000,B 0.000,C 90.000,E1 317.229} C_DIS
LIN {X -0.028,Y -212.041,Z 1821.749,A 0.000,B 0.000,C 90.000,E1 314.879} C_DIS
LIN {X -0.016,Y -215.891,Z 1821.740,A 0.000,B 0.000,C 90.000,E1 313.299} C_DIS
LIN {X -0.089,Y -220.421,Z 1821.732,A 0.000,B 0.000,C 90.000,E1 311.757} C_DIS
LIN {X 0.137,Y -224.332,Z 1821.725,A 0.000,B 0.000,C 90.000,E1 310.539} C_DIS
LIN {X 0.025,Y -230.213,Z 1821.717,A 0.000,B 0.000,C 90.000,E1 309.036} C_DIS
LIN {X -0.020,Y -238.612,Z 1821.706,A 0.000,B 0.000,C 90.000,E1 307.156} C_DIS
LIN {X -0.069,Y -247.887,Z 1821.696,A 0.000,B 0.000,C 90.000,E1 305.311} C_DIS
LIN {X 0.119,Y -260.113,Z 1821.684,A 0.000,B 0.000,C 90.000,E1 303.086} C_DIS
LIN {X 0.136,Y -278.255,Z 1821.668,A 0.000,B 0.000,C 90.000,E1 300.256} C_DIS
LIN {X -0.018,Y -292.782,Z 1821.657,A 0.000,B 0.000,C 90.000,E1 298.231} C_DIS
LIN {X -0.019,Y -310.152,Z 1821.644,A 0.000,B 0.000,C 90.000,E1 295.899} C_DIS
LIN {X 0.022,Y -325.235,Z 1821.633,A 0.000,B 0.000,C 90.000,E1 293.951} C_DIS
LIN {X -0.059,Y -337.578,Z 1821.624,A 0.000,B 0.000,C 90.000,E1 292.386} C_DIS
LIN {X -0.095,Y -347.132,Z 1821.617,A 0.000,B 0.000,C 90.000,E1 291.153} C_DIS
LIN {X -0.172,Y -353.980,Z 1821.612,A 0.000,B 0.000,C 90.000,E1 290.248} C_DIS
LIN {X -0.053,Y -360.280,Z 1821.607,A 0.000,B 0.000,C 90.000,E1 289.322} C_DIS
LIN {X 0.000,Y -366.037,Z 1821.602,A 0.000,B 0.000,C 90.000,E1 288.417} C_DIS
LIN {X 0.115,Y -371.027,Z 1821.597,A 0.000,B 0.000,C 90.000,E1 287.511} C_DIS
LIN {X 0.181,Y -373.876,Z 1821.594,A 0.000,B 0.000,C 90.000,E1 286.913} C_DIS
LIN {X -0.101,Y -377.420,Z 1821.589,A 0.000,B 0.000,C 90.000,E1 286.079} C_DIS
LIN {X 0.007,Y -379.352,Z 1821.586,A 0.000,B 0.000,C 90.000,E1 285.481} C_DIS
LIN {X 0.023,Y -380.909,Z 1821.583,A 0.000,B 0.000,C 90.000,E1 284.898} C_DIS
LIN {X 0.150,Y -382.113,Z 1821.580,A 0.000,B 0.000,C 90.000,E1 284.300} C_DIS
LIN {X -0.178,Y -382.906,Z 1821.576,A 0.000,B 0.000,C 90.000,E1 283.772} C_DIS
LIN {X -0.038,Y -383.290,Z 1821.573,A 0.000,B 0.000,C 90.000,E1 283.175} C_DIS
LIN {X 0.017,Y -383.198,Z 1821.570,A 0.000,B 0.000,C 90.000,E1 282.591} C_DIS
LIN {X 0.077,Y -382.714,Z 1821.567,A 0.000,B 0.000,C 90.000,E1 282.007} C_DIS
LIN {X 0.138,Y -381.798,Z 1821.564,A 0.000,B 0.000,C 90.000,E1 281.422} C_DIS
LIN {X -0.179,Y -380.457,Z 1821.560,A 0.000,B 0.000,C 90.000,E1 280.894} C_DIS
LIN {X -0.128,Y -378.689,Z 1821.557,A 0.000,B 0.000,C 90.000,E1 280.310} C_DIS
LIN {X -0.072,Y -375.468,Z 1821.552,A 0.000,B 0.000,C 90.000,E1 279.434} C_DIS
LIN {X -0.112,Y -370.453,Z 1821.546,A 0.000,B 0.000,C 90.000,E1 278.276} C_DIS
LIN {X 0.172,Y -366.178,Z 1821.541,A 0.000,B 0.000,C 90.000,E1 277.352} C_DIS
LIN {X 0.047,Y -361.181,Z 1821.536,A 0.000,B 0.000,C 90.000,E1 276.486} C_DIS
LIN {X -0.069,Y -357.356,Z 1821.533,A 0.000,B 0.000,C 90.000,E1 275.910} C_DIS
LIN {X 0.147,Y -352.963,Z 1821.529,A 0.000,B 0.000,C 90.000,E1 275.277} C_DIS
LIN {X -0.015,Y -347.918,Z 1821.526,A 0.000,B 0.000,C 90.000,E1 274.702} C_DIS
LIN {X -0.137,Y -342.314,Z 1821.523,A 0.000,B 0.000,C 90.000,E1 274.131} C_DIS
LIN {X -0.047,Y -336.422,Z 1821.520,A 0.000,B 0.000,C 90.000,E1 273.555} C_DIS
LIN {X -0.060,Y -330.264,Z 1821.517,A 0.000,B 0.000,C 90.000,E1 273.037} C_DIS
LIN {X -0.148,Y -323.903,Z 1821.514,A 0.000,B 0.000,C 90.000,E1 272.579} C_DIS
LIN {X 0.060,Y -317.385,Z 1821.512,A 0.000,B 0.000,C 90.000,E1 272.121} C_DIS
LIN {X -0.084,Y -310.517,Z 1821.510,A 0.000,B 0.000,C 90.000,E1 271.776} C_DIS
LIN {X 0.023,Y -303.213,Z 1821.508,A 0.000,B 0.000,C 90.000,E1 271.432} C_DIS
LIN {X 0.108,Y -295.764,Z 1821.506,A 0.000,B 0.000,C 90.000,E1 271.146} C_DIS
LIN {X -0.115,Y -288.025,Z 1821.505,A 0.000,B 0.000,C 90.000,E1 270.974} C_DIS
LIN {X 0.064,Y -276.560,Z 1821.504,A 0.000,B 0.000,C 90.000,E1 270.688} C_DIS
LIN {X 0.001,Y -250.807,Z 1821.501,A 0.000,B 0.000,C 90.000,E1 270.229} C_DIS
LIN {X -0.032,Y -240.560,Z 1821.501,A 0.000,B 0.000,C 90.000,E1 270.115} C_DIS
LIN {X 0.036,Y -232.716,Z 1821.500,A 0.000,B 0.000,C 90.000,E1 270.057} C_DIS
LIN {X 0.002,Y -181.569,Z 1821.500,A 0.000,B 0.000,C 90.000,E1 270.057} C_DIS
LIN {X 0.086,Y -180.907,Z 1821.475,A 0.000,B 0.000,C 90.000,E1 265.469} C_DIS
LIN {X -0.036,Y -180.748,Z 1821.470,A 0.000,B 0.000,C 90.000,E1 264.666} C_DIS
LIN {X 0.032,Y -178.840,Z 1821.442,A 0.000,B 0.000,C 90.000,E1 259.577} C_DIS
LIN {X -0.071,Y -175.883,Z 1821.414,A 0.000,B 0.000,C 90.000,E1 254.519} C_DIS
LIN {X 0.035,Y -174.550,Z 1821.404,A 0.000,B 0.000,C 90.000,E1 252.779} C_DIS
LIN {X -0.033,Y -171.534,Z 1821.381,A 0.000,B 0.000,C 90.000,E1 248.518} C_DIS
LIN {X -0.040,Y -167.759,Z 1821.357,A 0.000,B 0.000,C 90.000,E1 244.204} C_DIS
LIN {X -0.098,Y -166.464,Z 1821.347,A 0.000,B 0.000,C 90.000,E1 242.487} C_DIS
LIN {X 0.040,Y -163.179,Z 1821.328,A 0.000,B 0.000,C 90.000,E1 238.948} C_DIS
LIN {X -0.045,Y -161.139,Z 1821.313,A 0.000,B 0.000,C 90.000,E1 236.342} C_DIS
LIN {X -0.009,Y -157.159,Z 1821.288,A 0.000,B 0.000,C 90.000,E1 231.904} C_DIS
LIN {X 0.014,Y -155.891,Z 1821.278,A 0.000,B 0.000,C 90.000,E1 230.114} C_DIS
LIN {X -0.028,Y -152.141,Z 1821.254,A 0.000,B 0.000,C 90.000,E1 225.648} C_DIS
LIN {X -0.007,Y -150.391,Z 1821.239,A 0.000,B 0.000,C 90.000,E1 222.933} C_DIS
LIN {X 0.016,Y -147.122,Z 1821.213,A 0.000,B 0.000,C 90.000,E1 218.382} C_DIS
LIN {X 0.007,Y -145.686,Z 1821.198,A 0.000,B 0.000,C 90.000,E1 215.644} C_DIS
LIN {X 0.004,Y -143.068,Z 1821.172,A 0.000,B 0.000,C 90.000,E1 211.052} C_DIS
LIN {X -0.064,Y -141.689,Z 1821.152,A 0.000,B 0.000,C 90.000,E1 207.385} C_DIS
LIN {X -0.010,Y -139.461,Z 1821.116,A 0.000,B 0.000,C 90.000,E1 200.865} C_DIS
LIN {X -0.041,Y -139.195,Z 1821.106,A 0.000,B 0.000,C 90.000,E1 199.014} C_DIS
LIN {X -0.023,Y -138.325,Z 1821.054,A 0.000,B 0.000,C 90.000,E1 189.670} C_DIS
LIN {X -0.018,Y -139.451,Z 1821.007,A 0.000,B 0.000,C 90.000,E1 181.260} C_DIS
LIN {X 0.062,Y -140.996,Z 1820.976,A 0.000,B 0.000,C 90.000,E1 175.641} C_DIS
LIN {X 0.012,Y -142.751,Z 1820.955,A 0.000,B 0.000,C 90.000,E1 171.951} C_DIS
LIN {X -0.031,Y -145.150,Z 1820.930,A 0.000,B 0.000,C 90.000,E1 167.353} C_DIS
LIN {X -0.039,Y -147.774,Z 1820.909,A 0.000,B 0.000,C 90.000,E1 163.685} C_DIS
LIN {X 0.041,Y -150.450,Z 1820.889,A 0.000,B 0.000,C 90.000,E1 160.007} C_DIS
LIN {X -0.025,Y -153.897,Z 1820.869,A 0.000,B 0.000,C 90.000,E1 156.410} C_DIS
LIN {X 0.041,Y -157.307,Z 1820.849,A 0.000,B 0.000,C 90.000,E1 152.794} C_DIS
LIN {X -0.013,Y -161.494,Z 1820.829,A 0.000,B 0.000,C 90.000,E1 149.253} C_DIS
LIN {X 0.003,Y -165.693,Z 1820.810,A 0.000,B 0.000,C 90.000,E1 145.722} C_DIS
LIN {X -0.111,Y -170.636,Z 1820.790,A 0.000,B 0.000,C 90.000,E1 142.271} C_DIS
LIN {X 0.043,Y -175.511,Z 1820.771,A 0.000,B 0.000,C 90.000,E1 138.771} C_DIS
LIN {X -0.092,Y -181.132,Z 1820.752,A 0.000,B 0.000,C 90.000,E1 135.405} C_DIS
LIN {X 0.035,Y -186.582,Z 1820.733,A 0.000,B 0.000,C 90.000,E1 132.000} C_DIS
LIN {X -0.016,Y -191.194,Z 1820.719,A 0.000,B 0.000,C 90.000,E1 129.519} C_DIS
LIN {X 0.030,Y -197.003,Z 1820.701,A 0.000,B 0.000,C 90.000,E1 126.217} C_DIS
LIN {X -0.051,Y -200.272,Z 1820.692,A 0.000,B 0.000,C 90.000,E1 124.612} C_DIS
LIN {X -0.059,Y -207.764,Z 1820.670,A 0.000,B 0.000,C 90.000,E1 120.590} C_DIS
LIN {X -0.056,Y -210.939,Z 1820.661,A 0.000,B 0.000,C 90.000,E1 118.999} C_DIS
LIN {X -0.050,Y -216.809,Z 1820.644,A 0.000,B 0.000,C 90.000,E1 115.848} C_DIS
LIN {X 0.098,Y -218.425,Z 1820.639,A 0.000,B 0.000,C 90.000,E1 115.027} C_DIS
LIN {X -0.062,Y -221.151,Z 1820.630,A 0.000,B 0.000,C 90.000,E1 113.515} C_DIS
LIN {X -0.032,Y -224.026,Z 1820.622,A 0.000,B 0.000,C 90.000,E1 111.897} C_DIS
LIN {X -0.076,Y -283.708,Z 1820.622,A 0.000,B 0.000,C 90.000,E1 111.897} C_DIS
LIN {X -0.098,Y -288.714,Z 1820.620,A 0.000,B 0.000,C 90.000,E1 111.716} C_DIS
LIN {X -0.049,Y -290.960,Z 1820.620,A 0.000,B 0.000,C 90.000,E1 111.535} C_DIS
LIN {X 0.054,Y -294.038,Z 1820.618,A 0.000,B 0.000,C 90.000,E1 111.173} C_DIS
LIN {X 0.053,Y -296.045,Z 1820.616,A 0.000,B 0.000,C 90.000,E1 110.865} C_DIS
LIN {X -0.102,Y -309.110,Z 1820.603,A 0.000,B 0.000,C 90.000,E1 108.598} C_DIS
LIN {X -0.011,Y -323.659,Z 1820.591,A 0.000,B 0.000,C 90.000,E1 106.315} C_DIS
LIN {X 0.032,Y -337.315,Z 1820.580,A 0.000,B 0.000,C 90.000,E1 104.411} C_DIS
LIN {X -0.163,Y -352.152,Z 1820.570,A 0.000,B 0.000,C 90.000,E1 102.591} C_DIS
LIN {X -0.179,Y -370.546,Z 1820.558,A 0.000,B 0.000,C 90.000,E1 100.546} C_DIS
LIN {X -0.136,Y -389.363,Z 1820.548,A 0.000,B 0.000,C 90.000,E1 98.681} C_DIS
LIN {X 0.138,Y -408.599,Z 1820.539,A 0.000,B 0.000,C 90.000,E1 96.947} C_DIS
LIN {X -0.061,Y -430.962,Z 1820.529,A 0.000,B 0.000,C 90.000,E1 95.220} C_DIS
LIN {X 0.096,Y -439.343,Z 1820.526,A 0.000,B 0.000,C 90.000,E1 94.588} C_DIS
LIN {X -0.129,Y -441.461,Z 1820.524,A 0.000,B 0.000,C 90.000,E1 94.416} C_DIS
LIN {X 0.185,Y -443.421,Z 1820.523,A 0.000,B 0.000,C 90.000,E1 94.131} C_DIS
LIN {X 0.090,Y -444.921,Z 1820.522,A 0.000,B 0.000,C 90.000,E1 93.898} C_DIS
LIN {X -0.175,Y -446.149,Z 1820.520,A 0.000,B 0.000,C 90.000,E1 93.669} C_DIS
LIN {X 0.005,Y -447.056,Z 1820.519,A 0.000,B 0.000,C 90.000,E1 93.383} C_DIS
LIN {X -0.039,Y -448.065,Z 1820.516,A 0.000,B 0.000,C 90.000,E1 92.865} C_DIS
LIN {X -0.100,Y -448.126,Z 1820.513,A 0.000,B 0.000,C 90.000,E1 92.350} C_DIS
LIN {X -0.152,Y -447.249,Z 1820.510,A 0.000,B 0.000,C 90.000,E1 91.835} C_DIS
LIN {X -0.190,Y -445.298,Z 1820.507,A 0.000,B 0.000,C 90.000,E1 91.318} C_DIS
LIN {X -0.061,Y -440.493,Z 1820.503,A 0.000,B 0.000,C 90.000,E1 90.516} C_DIS
LIN {X -0.215,Y -428.959,Z 1820.493,A 0.000,B 0.000,C 90.000,E1 88.682} C_DIS
LIN {X -0.150,Y -417.199,Z 1820.482,A 0.000,B 0.000,C 90.000,E1 86.788} C_DIS
LIN {X 0.021,Y -407.069,Z 1820.473,A 0.000,B 0.000,C 90.000,E1 85.122} C_DIS
LIN {X 0.073,Y -395.158,Z 1820.462,A 0.000,B 0.000,C 90.000,E1 83.166} C_DIS
LIN {X -0.034,Y -383.203,Z 1820.451,A 0.000,B 0.000,C 90.000,E1 81.197} C_DIS
LIN {X 0.055,Y -369.604,Z 1820.438,A 0.000,B 0.000,C 90.000,E1 78.870} C_DIS
LIN {X -0.177,Y -351.833,Z 1820.420,A 0.000,B 0.000,C 90.000,E1 75.644} C_DIS
LIN {X -0.184,Y -338.145,Z 1820.405,A 0.000,B 0.000,C 90.000,E1 72.906} C_DIS
LIN {X 0.127,Y -327.767,Z 1820.393,A 0.000,B 0.000,C 90.000,E1 70.678} C_DIS
LIN {X -0.075,Y -313.400,Z 1820.375,A 0.000,B 0.000,C 90.000,E1 67.539} C_DIS
LIN {X 0.138,Y -303.757,Z 1820.363,A 0.000,B 0.000,C 90.000,E1 65.229} C_DIS
LIN {X -0.012,Y -292.816,Z 1820.348,A 0.000,B 0.000,C 90.000,E1 62.615} C_DIS
LIN {X 0.037,Y -284.835,Z 1820.337,A 0.000,B 0.000,C 90.000,E1 60.589} C_DIS
LIN {X -0.105,Y -278.261,Z 1820.327,A 0.000,B 0.000,C 90.000,E1 58.948} C_DIS
LIN {X -0.014,Y -278.257,Z 1820.327,A 0.000,B 0.000,C 90.000,E1 58.918} C_DIS
LIN {X -0.073,Y -283.898,Z 1820.320,A 0.000,B 0.000,C 90.000,E1 57.533} C_DIS
LIN {X 0.003,Y -284.981,Z 1820.316,A 0.000,B 0.000,C 90.000,E1 56.834} C_DIS
LIN {X -0.067,Y -284.597,Z 1820.312,A 0.000,B 0.000,C 90.000,E1 56.167} C_DIS
LIN {X 0.027,Y -283.673,Z 1820.308,A 0.000,B 0.000,C 90.000,E1 55.468} C_DIS
LIN {X 0.118,Y -282.434,Z 1820.304,A 0.000,B 0.000,C 90.000,E1 54.769} C_DIS
LIN {X 0.054,Y -279.458,Z 1820.297,A 0.000,B 0.000,C 90.000,E1 53.417} C_DIS
LIN {X -0.047,Y -276.029,Z 1820.289,A 0.000,B 0.000,C 90.000,E1 52.065} C_DIS
LIN {X -0.043,Y -270.519,Z 1820.278,A 0.000,B 0.000,C 90.000,E1 49.989} C_DIS
LIN {X 0.030,Y -264.760,Z 1820.266,A 0.000,B 0.000,C 90.000,E1 47.877} C_DIS
LIN {X 0.152,Y -258.951,Z 1820.254,A 0.000,B 0.000,C 90.000,E1 45.729} C_DIS
LIN {X 0.021,Y -251.113,Z 1820.238,A 0.000,B 0.000,C 90.000,E1 42.894} C_DIS
LIN {X 0.088,Y -245.167,Z 1820.226,A 0.000,B 0.000,C 90.000,E1 40.701} C_DIS
LIN {X -0.132,Y -237.236,Z 1820.210,A 0.000,B 0.000,C 90.000,E1 37.810} C_DIS
LIN {X 0.086,Y -231.277,Z 1820.197,A 0.000,B 0.000,C 90.000,E1 35.518} C_DIS
LIN {X 0.051,Y -223.473,Z 1820.181,A 0.000,B 0.000,C 90.000,E1 32.498} C_DIS
LIN {X 0.084,Y -215.861,Z 1820.164,A 0.000,B 0.000,C 90.000,E1 29.411} C_DIS
LIN {X -0.008,Y -208.989,Z 1820.146,A 0.000,B 0.000,C 90.000,E1 26.309} C_DIS
LIN {X 0.010,Y -202.818,Z 1820.129,A 0.000,B 0.000,C 90.000,E1 23.131} C_DIS
LIN {X -0.069,Y -197.707,Z 1820.111,A 0.000,B 0.000,C 90.000,E1 19.939} C_DIS
LIN {X -0.029,Y -193.406,Z 1820.093,A 0.000,B 0.000,C 90.000,E1 16.677} C_DIS
LIN {X -0.091,Y -189.028,Z 1820.070,A 0.000,B 0.000,C 90.000,E1 12.591} C_DIS
LIN {X 0.070,Y -185.699,Z 1820.047,A 0.000,B 0.000,C 90.000,E1 8.398} C_DIS
LIN {X -0.030,Y -182.602,Z 1820.014,A 0.000,B 0.000,C 90.000,E1 2.579} C_DIS
LIN {X -0.024,Y -181.273,Z 1819.969,A 0.000,B 0.000,C 90.000,E1 354.489} C_DIS
LIN {X -0.036,Y -182.162,Z 1819.932,A 0.000,B 0.000,C 90.000,E1 347.757} C_DIS
LIN {X -0.057,Y -183.816,Z 1819.904,A 0.000,B 0.000,C 90.000,E1 342.725} C_DIS
LIN {X -0.042,Y -186.912,Z 1819.871,A 0.000,B 0.000,C 90.000,E1 336.869} C_DIS
LIN {X -0.068,Y -190.432,Z 1819.844,A 0.000,B 0.000,C 90.000,E1 331.897} C_DIS
LIN {X -0.099,Y -194.022,Z 1819.821,A 0.000,B 0.000,C 90.000,E1 327.788} C_DIS
LIN {X -0.099,Y -198.122,Z 1819.798,A 0.000,B 0.000,C 90.000,E1 323.703} C_DIS
LIN {X -0.007,Y -202.173,Z 1819.780,A 0.000,B 0.000,C 90.000,E1 320.436} C_DIS
LIN {X 0.086,Y -205.865,Z 1819.767,A 0.000,B 0.000,C 90.000,E1 318.000} C_DIS
LIN {X 0.030,Y -208.751,Z 1819.758,A 0.000,B 0.000,C 90.000,E1 316.419} C_DIS
LIN {X 0.008,Y -212.110,Z 1819.749,A 0.000,B 0.000,C 90.000,E1 314.838} C_DIS
LIN {X 0.027,Y -216.018,Z 1819.740,A 0.000,B 0.000,C 90.000,E1 313.257} C_DIS
LIN {X 0.107,Y -220.580,Z 1819.732,A 0.000,B 0.000,C 90.000,E1 311.676} C_DIS
LIN {X -0.051,Y -225.942,Z 1819.723,A 0.000,B 0.000,C 90.000,E1 310.172} C_DIS
LIN {X 0.032,Y -232.072,Z 1819.715,A 0.000,B 0.000,C 90.000,E1 308.624} C_DIS
LIN {X 0.028,Y -240.664,Z 1819.704,A 0.000,B 0.000,C 90.000,E1 306.744} C_DIS
LIN {X 0.014,Y -252.188,Z 1819.692,A 0.000,B 0.000,C 90.000,E1 304.532} C_DIS
LIN {X -0.113,Y -262.680,Z 1819.682,A 0.000,B 0.000,C 90.000,E1 302.752} C_DIS
LIN {X -0.042,Y -281.089,Z 1819.666,A 0.000,B 0.000,C 90.000,E1 299.922} C_DIS
LIN {X 0.110,Y -295.674,Z 1819.655,A 0.000,B 0.000,C 90.000,E1 297.847} C_DIS
LIN {X 0.055,Y -313.201,Z 1819.642,A 0.000,B 0.000,C 90.000,E1 295.540} C_DIS
LIN {X -0.080,Y -325.799,Z 1819.633,A 0.000,B 0.000,C 90.000,E1 293.951} C_DIS
LIN {X 0.158,Y -338.184,Z 1819.624,A 0.000,B 0.000,C 90.000,E1 292.333} C_DIS
LIN {X 0.138,Y -347.770,Z 1819.617,A 0.000,B 0.000,C 90.000,E1 291.099} C_DIS
LIN {X 0.074,Y -354.644,Z 1819.612,A 0.000,B 0.000,C 90.000,E1 290.194} C_DIS
LIN {X -0.135,Y -360.930,Z 1819.607,A 0.000,B 0.000,C 90.000,E1 289.322} C_DIS
LIN {X -0.077,Y -366.679,Z 1819.602,A 0.000,B 0.000,C 90.000,E1 288.417} C_DIS
LIN {X 0.044,Y -371.649,Z 1819.597,A 0.000,B 0.000,C 90.000,E1 287.511} C_DIS
LIN {X 0.113,Y -374.460,Z 1819.594,A 0.000,B 0.000,C 90.000,E1 286.913} C_DIS
LIN {X 0.202,Y -376.937,Z 1819.591,A 0.000,B 0.000,C 90.000,E1 286.315} C_DIS
LIN {X -0.054,Y -379.931,Z 1819.586,A 0.000,B 0.000,C 90.000,E1 285.481} C_DIS
LIN {X -0.034,Y -381.469,Z 1819.583,A 0.000,B 0.000,C 90.000,E1 284.898} C_DIS
LIN {X 0.097,Y -382.662,Z 1819.579,A 0.000,B 0.000,C 90.000,E1 284.300} C_DIS
LIN {X 0.144,Y -383.431,Z 1819.576,A 0.000,B 0.000,C 90.000,E1 283.716} C_DIS
LIN {X -0.086,Y -383.802,Z 1819.573,A 0.000,B 0.000,C 90.000,E1 283.175} C_DIS
LIN {X -0.027,Y -383.722,Z 1819.570,A 0.000,B 0.000,C 90.000,E1 282.591} C_DIS
LIN {X 0.037,Y -383.217,Z 1819.567,A 0.000,B 0.000,C 90.000,E1 282.007} C_DIS
LIN {X 0.100,Y -382.277,Z 1819.564,A 0.000,B 0.000,C 90.000,E1 281.422} C_DIS
LIN {X 0.160,Y -380.920,Z 1819.560,A 0.000,B 0.000,C 90.000,E1 280.838} C_DIS
LIN {X -0.159,Y -379.172,Z 1819.557,A 0.000,B 0.000,C 90.000,E1 280.310} C_DIS
LIN {X -0.099,Y -375.977,Z 1819.552,A 0.000,B 0.000,C 90.000,E1 279.434} C_DIS
LIN {X -0.133,Y -370.969,Z 1819.546,A 0.000,B 0.000,C 90.000,E1 278.276} C_DIS
LIN {X 0.156,Y -366.636,Z 1819.541,A 0.000,B 0.000,C 90.000,E1 277.352} C_DIS
LIN {X 0.037,Y -361.555,Z 1819.536,A 0.000,B 0.000,C 90.000,E1 276.486} C_DIS
LIN {X -0.157,Y -355.566,Z 1819.531,A 0.000,B 0.000,C 90.000,E1 275.625} C_DIS
LIN {X 0.052,Y -350.781,Z 1819.528,A 0.000,B 0.000,C 90.000,E1 274.992} C_DIS
LIN {X -0.117,Y -345.390,Z 1819.524,A 0.000,B 0.000,C 90.000,E1 274.416} C_DIS
LIN {X -0.163,Y -339.522,Z 1819.521,A 0.000,B 0.000,C 90.000,E1 273.841} C_DIS
LIN {X 0.030,Y -333.459,Z 1819.518,A 0.000,B 0.000,C 90.000,E1 273.269} C_DIS
LIN {X -0.150,Y -327.219,Z 1819.516,A 0.000,B 0.000,C 90.000,E1 272.808} C_DIS
LIN {X -0.092,Y -320.815,Z 1819.513,A 0.000,B 0.000,C 90.000,E1 272.350} C_DIS
LIN {X -0.095,Y -314.063,Z 1819.511,A 0.000,B 0.000,C 90.000,E1 271.949} C_DIS
LIN {X -0.114,Y -306.972,Z 1819.509,A 0.000,B 0.000,C 90.000,E1 271.604} C_DIS
LIN {X -0.140,Y -299.623,Z 1819.507,A 0.000,B 0.000,C 90.000,E1 271.318} C_DIS
LIN {X 0.102,Y -291.940,Z 1819.506,A 0.000,B 0.000,C 90.000,E1 271.031} C_DIS
LIN {X -0.067,Y -280.907,Z 1819.504,A 0.000,B 0.000,C 90.000,E1 270.802} C_DIS
LIN {X 0.110,Y -255.429,Z 1819.502,A 0.000,B 0.000,C 90.000,E1 270.286} C_DIS
LIN {X 0.025,Y -246.755,Z 1819.501,A 0.000,B 0.000,C 90.000,E1 270.172} C_DIS
LIN {X -0.092,Y -236.942,Z 1819.500,A 0.000,B 0.000,C 90.000,E1 270.115} C_DIS
LIN {X 0.077,Y -232.555,Z 1819.500,A 0.000,B 0.000,C 90.000,E1 270.057} C_DIS
LIN {X 0.034,Y -181.570,Z 1819.500,A 0.000,B 0.000,C 90.000,E1 270.057} C_DIS
LIN {X -0.037,Y -180.907,Z 1819.475,A 0.000,B 0.000,C 90.000,E1 265.527} C_DIS
LIN {X 0.020,Y -180.756,Z 1819.470,A 0.000,B 0.000,C 90.000,E1 264.666} C_DIS
LIN {X -0.087,Y -178.849,Z 1819.442,A 0.000,B 0.000,C 90.000,E1 259.634} C_DIS
LIN {X -0.016,Y -175.892,Z 1819.414,A 0.000,B 0.000,C 90.000,E1 254.519} C_DIS
LIN {X 0.090,Y -174.565,Z 1819.405,A 0.000,B 0.000,C 90.000,E1 252.779} C_DIS
LIN {X -0.041,Y -171.548,Z 1819.381,A 0.000,B 0.000,C 90.000,E1 248.539} C_DIS
LIN {X 0.015,Y -167.772,Z 1819.357,A 0.000,B 0.000,C 90.000,E1 244.204} C_DIS
LIN {X -0.043,Y -166.482,Z 1819.347,A 0.000,B 0.000,C 90.000,E1 242.487} C_DIS
LIN {X -0.047,Y -163.194,Z 1819.328,A 0.000,B 0.000,C 90.000,E1 238.997} C_DIS
LIN {X 0.008,Y -161.157,Z 1819.313,A 0.000,B 0.000,C 90.000,E1 236.342} C_DIS
LIN {X 0.043,Y -157.174,Z 1819.288,A 0.000,B 0.000,C 90.000,E1 231.904} C_DIS
LIN {X -0.034,Y -155.905,Z 1819.279,A 0.000,B 0.000,C 90.000,E1 230.150} C_DIS
LIN {X 0.023,Y -152.155,Z 1819.254,A 0.000,B 0.000,C 90.000,E1 225.648} C_DIS
LIN {X 0.043,Y -150.405,Z 1819.239,A 0.000,B 0.000,C 90.000,E1 222.933} C_DIS
LIN {X 0.066,Y -147.134,Z 1819.213,A 0.000,B 0.000,C 90.000,E1 218.382} C_DIS
LIN {X -0.028,Y -145.695,Z 1819.198,A 0.000,B 0.000,C 90.000,E1 215.678} C_DIS
LIN {X 0.053,Y -143.078,Z 1819.173,A 0.000,B 0.000,C 90.000,E1 211.052} C_DIS
LIN {X -0.015,Y -141.696,Z 1819.152,A 0.000,B 0.000,C 90.000,E1 207.385} C_DIS
LIN {X 0.039,Y -139.464,Z 1819.116,A 0.000,B 0.000,C 90.000,E1 200.865} C_DIS
LIN {X -0.037,Y -139.198,Z 1819.106,A 0.000,B 0.000,C 90.000,E1 199.033} C_DIS
LIN {X 0.025,Y -138.326,Z 1819.054,A 0.000,B 0.000,C 90.000,E1 189.670} C_DIS
LIN {X 0.031,Y -139.447,Z 1819.007,A 0.000,B 0.000,C 90.000,E1 181.260} C_DIS
LIN {X -0.029,Y -140.988,Z 1818.976,A 0.000,B 0.000,C 90.000,E1 175.698} C_DIS
LIN {X 0.062,Y -142.743,Z 1818.955,A 0.000,B 0.000,C 90.000,E1 171.951} C_DIS
LIN {X 0.018,Y -145.138,Z 1818.930,A 0.000,B 0.000,C 90.000,E1 167.353} C_DIS
LIN {X 0.012,Y -147.761,Z 1818.909,A 0.000,B 0.000,C 90.000,E1 163.685} C_DIS
LIN {X -0.050,Y -150.434,Z 1818.889,A 0.000,B 0.000,C 90.000,E1 160.061} C_DIS
LIN {X -0.035,Y -153.878,Z 1818.869,A 0.000,B 0.000,C 90.000,E1 156.433} C_DIS
LIN {X 0.021,Y -157.288,Z 1818.849,A 0.000,B 0.000,C 90.000,E1 152.820} C_DIS
LIN {X -0.042,Y -161.469,Z 1818.829,A 0.000,B 0.000,C 90.000,E1 149.282} C_DIS
LIN {X -0.037,Y -165.669,Z 1818.810,A 0.000,B 0.000,C 90.000,E1 145.754} C_DIS
LIN {X -0.055,Y -170.607,Z 1818.790,A 0.000,B 0.000,C 90.000,E1 142.271} C_DIS
LIN {X 0.099,Y -175.484,Z 1818.771,A 0.000,B 0.000,C 90.000,E1 138.771} C_DIS
LIN {X -0.035,Y -181.106,Z 1818.752,A 0.000,B 0.000,C 90.000,E1 135.405} C_DIS
LIN {X -0.045,Y -186.550,Z 1818.734,A 0.000,B 0.000,C 90.000,E1 132.043} C_DIS
LIN {X -0.104,Y -191.165,Z 1818.720,A 0.000,B 0.000,C 90.000,E1 129.564} C_DIS
LIN {X 0.090,Y -196.970,Z 1818.701,A 0.000,B 0.000,C 90.000,E1 126.217} C_DIS
LIN {X 0.009,Y -200.236,Z 1818.692,A 0.000,B 0.000,C 90.000,E1 124.612} C_DIS
LIN {X 0.004,Y -207.729,Z 1818.670,A 0.000,B 0.000,C 90.000,E1 120.590} C_DIS
LIN {X 0.006,Y -210.909,Z 1818.661,A 0.000,B 0.000,C 90.000,E1 118.999} C_DIS
LIN {X 0.013,Y -216.775,Z 1818.644,A 0.000,B 0.000,C 90.000,E1 115.848} C_DIS
LIN {X 0.032,Y -219.829,Z 1818.635,A 0.000,B 0.000,C 90.000,E1 114.283} C_DIS
LIN {X -0.024,Y -224.022,Z 1818.622,A 0.000,B 0.000,C 90.000,E1 111.897} C_DIS
LIN {X -0.065,Y -283.663,Z 1818.622,A 0.000,B 0.000,C 90.000,E1 111.897} C_DIS
LIN {X -0.017,Y -288.468,Z 1818.621,A 0.000,B 0.000,C 90.000,E1 111.716} C_DIS
LIN {X 0.035,Y -290.784,Z 1818.620,A 0.000,B 0.000,C 90.000,E1 111.535} C_DIS
LIN {X -0.136,Y -293.919,Z 1818.618,A 0.000,B 0.000,C 90.000,E1 111.227} C_DIS
LIN {X -0.119,Y -295.927,Z 1818.616,A 0.000,B 0.000,C 90.000,E1 110.918} C_DIS
LIN {X 0.028,Y -308.962,Z 1818.603,A 0.000,B 0.000,C 90.000,E1 108.598} C_DIS
LIN {X 0.123,Y -323.497,Z 1818.591,A 0.000,B 0.000,C 90.000,E1 106.315} C_DIS
LIN {X 0.083,Y -337.138,Z 1818.580,A 0.000,B 0.000,C 90.000,E1 104.426} C_DIS
LIN {X -0.025,Y -351.961,Z 1818.570,A 0.000,B 0.000,C 90.000,E1 102.591} C_DIS
LIN {X -0.047,Y -370.348,Z 1818.559,A 0.000,B 0.000,C 90.000,E1 100.546} C_DIS
LIN {X -0.009,Y -389.162,Z 1818.548,A 0.000,B 0.000,C 90.000,E1 98.681} C_DIS
LIN {X -0.147,Y -408.394,Z 1818.539,A 0.000,B 0.000,C 90.000,E1 97.004} C_DIS
LIN {X 0.053,Y -430.754,Z 1818.529,A 0.000,B 0.000,C 90.000,E1 95.220} C_DIS
LIN {X 0.208,Y -439.159,Z 1818.526,A 0.000,B 0.000,C 90.000,E1 94.588} C_DIS
LIN {X -0.018,Y -441.320,Z 1818.525,A 0.000,B 0.000,C 90.000,E1 94.416} C_DIS
LIN {X -0.120,Y -443.290,Z 1818.523,A 0.000,B 0.000,C 90.000,E1 94.188} C_DIS
LIN {X -0.193,Y -444.800,Z 1818.522,A 0.000,B 0.000,C 90.000,E1 93.955} C_DIS
LIN {X -0.015,Y -446.054,Z 1818.520,A 0.000,B 0.000,C 90.000,E1 93.669} C_DIS
LIN {X 0.165,Y -446.985,Z 1818.519,A 0.000,B 0.000,C 90.000,E1 93.383} C_DIS
LIN {X 0.122,Y -448.031,Z 1818.516,A 0.000,B 0.000,C 90.000,E1 92.865} C_DIS
LIN {X 0.060,Y -448.126,Z 1818.513,A 0.000,B 0.000,C 90.000,E1 92.350} C_DIS
LIN {X 0.008,Y -447.287,Z 1818.510,A 0.000,B 0.000,C 90.000,E1 91.835} C_DIS
LIN {X -0.031,Y -445.382,Z 1818.507,A 0.000,B 0.000,C 90.000,E1 91.318} C_DIS
LIN {X -0.087,Y -442.258,Z 1818.504,A 0.000,B 0.000,C 90.000,E1 90.802} C_DIS
LIN {X -0.058,Y -429.071,Z 1818.493,A 0.000,B 0.000,C 90.000,E1 88.682} C_DIS
LIN {X 0.003,Y -417.311,Z 1818.482,A 0.000,B 0.000,C 90.000,E1 86.788} C_DIS
LIN {X 0.173,Y -407.182,Z 1818.473,A 0.000,B 0.000,C 90.000,E1 85.122} C_DIS
LIN {X -0.169,Y -395.273,Z 1818.462,A 0.000,B 0.000,C 90.000,E1 83.223} C_DIS
LIN {X 0.114,Y -383.319,Z 1818.451,A 0.000,B 0.000,C 90.000,E1 81.197} C_DIS
LIN {X 0.201,Y -369.714,Z 1818.438,A 0.000,B 0.000,C 90.000,E1 78.870} C_DIS
LIN {X -0.036,Y -351.934,Z 1818.420,A 0.000,B 0.000,C 90.000,E1 75.644} C_DIS
LIN {X -0.046,Y -338.240,Z 1818.405,A 0.000,B 0.000,C 90.000,E1 72.906} C_DIS
LIN {X -0.045,Y -327.859,Z 1818.393,A 0.000,B 0.000,C 90.000,E1 70.732} C_DIS
LIN {X 0.058,Y -313.484,Z 1818.375,A 0.000,B 0.000,C 90.000,E1 67.539} C_DIS
LIN {X -0.006,Y -303.839,Z 1818.363,A 0.000,B 0.000,C 90.000,E1 65.281} C_DIS
LIN {X 0.117,Y -292.895,Z 1818.348,A 0.000,B 0.000,C 90.000,E1 62.615} C_DIS
LIN {X -0.178,Y -285.461,Z 1818.338,A 0.000,B 0.000,C 90.000,E1 60.795} C_DIS
LIN {X 0.158,Y -285.437,Z 1818.338,A 0.000,B 0.000,C 90.000,E1 60.717} C_DIS
LIN {X -0.077,Y -291.180,Z 1818.329,A 0.000,B 0.000,C 90.000,E1 59.282} C_DIS
LIN {X -0.096,Y -292.218,Z 1818.327,A 0.000,B 0.000,C 90.000,E1 58.948} C_DIS
LIN {X 0.034,Y -292.437,Z 1818.324,A 0.000,B 0.000,C 90.000,E1 58.250} C_DIS
LIN {X 0.019,Y -291.754,Z 1818.320,A 0.000,B 0.000,C 90.000,E1 57.582} C_DIS
LIN {X 0.003,Y -290.671,Z 1818.316,A 0.000,B 0.000,C 90.000,E1 56.914} C_DIS
LIN {X 0.141,Y -289.319,Z 1818.313,A 0.000,B 0.000,C 90.000,E1 56.215} C_DIS
LIN {X -0.003,Y -286.115,Z 1818.305,A 0.000,B 0.000,C 90.000,E1 54.895} C_DIS
LIN {X -0.016,Y -282.504,Z 1818.297,A 0.000,B 0.000,C 90.000,E1 53.543} C_DIS
LIN {X 0.159,Y -276.650,Z 1818.286,A 0.000,B 0.000,C 90.000,E1 51.457} C_DIS
LIN {X 0.174,Y -270.595,Z 1818.275,A 0.000,B 0.000,C 90.000,E1 49.380} C_DIS
LIN {X -0.020,Y -262.405,Z 1818.259,A 0.000,B 0.000,C 90.000,E1 46.620} C_DIS
LIN {X -0.123,Y -256.259,Z 1818.247,A 0.000,B 0.000,C 90.000,E1 44.514} C_DIS
LIN {X 0.030,Y -250.109,Z 1818.235,A 0.000,B 0.000,C 90.000,E1 42.324} C_DIS
LIN {X -0.099,Y -243.924,Z 1818.223,A 0.000,B 0.000,C 90.000,E1 40.172} C_DIS
LIN {X -0.017,Y -235.707,Z 1818.207,A 0.000,B 0.000,C 90.000,E1 37.202} C_DIS
LIN {X 0.028,Y -229.474,Z 1818.194,A 0.000,B 0.000,C 90.000,E1 34.945} C_DIS
LIN {X -0.054,Y -221.540,Z 1818.177,A 0.000,B 0.000,C 90.000,E1 31.926} C_DIS
LIN {X 0.006,Y -214.055,Z 1818.160,A 0.000,B 0.000,C 90.000,E1 28.821} C_DIS
LIN {X 0.057,Y -207.304,Z 1818.143,A 0.000,B 0.000,C 90.000,E1 25.668} C_DIS
LIN {X -0.122,Y -202.706,Z 1818.129,A 0.000,B 0.000,C 90.000,E1 23.334} C_DIS
LIN {X 0.061,Y -197.516,Z 1818.112,A 0.000,B 0.000,C 90.000,E1 20.066} C_DIS
LIN {X -0.088,Y -193.168,Z 1818.094,A 0.000,B 0.000,C 90.000,E1 16.858} C_DIS
LIN {X 0.030,Y -188.752,Z 1818.071,A 0.000,B 0.000,C 90.000,E1 12.715} C_DIS
LIN {X 0.033,Y -185.390,Z 1818.048,A 0.000,B 0.000,C 90.000,E1 8.568} C_DIS
LIN {X 0.026,Y -182.616,Z 1818.020,A 0.000,B 0.000,C 90.000,E1 3.555} C_DIS
LIN {X 0.067,Y -180.922,Z 1817.974,A 0.000,B 0.000,C 90.000,E1 355.298} C_DIS
LIN {X -0.070,Y -181.781,Z 1817.932,A 0.000,B 0.000,C 90.000,E1 347.757} C_DIS
LIN {X -0.064,Y -183.807,Z 1817.899,A 0.000,B 0.000,C 90.000,E1 341.873} C_DIS
LIN {X -0.033,Y -186.582,Z 1817.871,A 0.000,B 0.000,C 90.000,E1 336.847} C_DIS
LIN {X 0.051,Y -189.505,Z 1817.848,A 0.000,B 0.000,C 90.000,E1 332.666} C_DIS
LIN {X -0.023,Y -193.767,Z 1817.821,A 0.000,B 0.000,C 90.000,E1 327.740} C_DIS
LIN {X 0.081,Y -197.924,Z 1817.798,A 0.000,B 0.000,C 90.000,E1 323.623} C_DIS
LIN {X -0.110,Y -202.053,Z 1817.780,A 0.000,B 0.000,C 90.000,E1 320.436} C_DIS
LIN {X -0.023,Y -205.825,Z 1817.767,A 0.000,B 0.000,C 90.000,E1 318.000} C_DIS
LIN {X 0.070,Y -208.769,Z 1817.758,A 0.000,B 0.000,C 90.000,E1 316.377} C_DIS
LIN {X -0.104,Y -212.178,Z 1817.749,A 0.000,B 0.000,C 90.000,E1 314.838} C_DIS
LIN {X 0.061,Y -216.158,Z 1817.740,A 0.000,B 0.000,C 90.000,E1 313.218} C_DIS
LIN {X -0.007,Y -220.764,Z 1817.732,A 0.000,B 0.000,C 90.000,E1 311.676} C_DIS
LIN {X -0.093,Y -224.723,Z 1817.725,A 0.000,B 0.000,C 90.000,E1 310.539} C_DIS
LIN {X -0.028,Y -230.715,Z 1817.717,A 0.000,B 0.000,C 90.000,E1 308.991} C_DIS
LIN {X 0.082,Y -239.154,Z 1817.706,A 0.000,B 0.000,C 90.000,E1 307.076} C_DIS
LIN {X 0.045,Y -248.546,Z 1817.696,A 0.000,B 0.000,C 90.000,E1 305.231} C_DIS
LIN {X -0.111,Y -260.888,Z 1817.684,A 0.000,B 0.000,C 90.000,E1 303.086} C_DIS
LIN {X -0.089,Y -279.113,Z 1817.668,A 0.000,B 0.000,C 90.000,E1 300.256} C_DIS
LIN {X 0.021,Y -293.717,Z 1817.657,A 0.000,B 0.000,C 90.000,E1 298.180} C_DIS
LIN {X 0.049,Y -311.177,Z 1817.644,A 0.000,B 0.000,C 90.000,E1 295.848} C_DIS
LIN {X -0.112,Y -323.862,Z 1817.635,A 0.000,B 0.000,C 90.000,E1 294.259} C_DIS
LIN {X 0.082,Y -336.371,Z 1817.626,A 0.000,B 0.000,C 90.000,E1 292.642} C_DIS
LIN {X 0.049,Y -348.387,Z 1817.617,A 0.000,B 0.000,C 90.000,E1 291.099} C_DIS
LIN {X 0.113,Y -355.258,Z 1817.612,A 0.000,B 0.000,C 90.000,E1 290.174} C_DIS
LIN {X 0.126,Y -361.608,Z 1817.607,A 0.000,B 0.000,C 90.000,E1 289.268} C_DIS
LIN {X -0.152,Y -367.322,Z 1817.602,A 0.000,B 0.000,C 90.000,E1 288.417} C_DIS
LIN {X -0.114,Y -370.739,Z 1817.599,A 0.000,B 0.000,C 90.000,E1 287.819} C_DIS
LIN {X -0.051,Y -373.758,Z 1817.596,A 0.000,B 0.000,C 90.000,E1 287.221} C_DIS
LIN {X 0.138,Y -377.528,Z 1817.591,A 0.000,B 0.000,C 90.000,E1 286.315} C_DIS
LIN {X -0.112,Y -380.497,Z 1817.586,A 0.000,B 0.000,C 90.000,E1 285.481} C_DIS
LIN {X -0.089,Y -382.016,Z 1817.583,A 0.000,B 0.000,C 90.000,E1 284.898} C_DIS
LIN {X 0.045,Y -383.175,Z 1817.579,A 0.000,B 0.000,C 90.000,E1 284.300} C_DIS
LIN {X 0.095,Y -383.948,Z 1817.576,A 0.000,B 0.000,C 90.000,E1 283.716} C_DIS
LIN {X -0.132,Y -384.295,Z 1817.573,A 0.000,B 0.000,C 90.000,E1 283.175} C_DIS
LIN {X -0.069,Y -384.237,Z 1817.570,A 0.000,B 0.000,C 90.000,E1 282.591} C_DIS
LIN {X -0.003,Y -383.683,Z 1817.567,A 0.000,B 0.000,C 90.000,E1 282.007} C_DIS
LIN {X 0.063,Y -382.751,Z 1817.563,A 0.000,B 0.000,C 90.000,E1 281.422} C_DIS
LIN {X 0.127,Y -381.421,Z 1817.560,A 0.000,B 0.000,C 90.000,E1 280.838} C_DIS
LIN {X 0.183,Y -379.720,Z 1817.557,A 0.000,B 0.000,C 90.000,E1 280.254} C_DIS
LIN {X -0.125,Y -376.512,Z 1817.552,A 0.000,B 0.000,C 90.000,E1 279.434} C_DIS
LIN {X -0.152,Y -371.509,Z 1817.546,A 0.000,B 0.000,C 90.000,E1 278.276} C_DIS
LIN {X 0.142,Y -367.120,Z 1817.541,A 0.000,B 0.000,C 90.000,E1 277.352} C_DIS
LIN {X 0.027,Y -361.951,Z 1817.536,A 0.000,B 0.000,C 90.000,E1 276.486} C_DIS
LIN {X -0.085,Y -358.021,Z 1817.533,A 0.000,B 0.000,C 90.000,E1 275.910} C_DIS
LIN {X 0.136,Y -353.559,Z 1817.529,A 0.000,B 0.000,C 90.000,E1 275.277} C_DIS
LIN {X -0.022,Y -348.407,Z 1817.526,A 0.000,B 0.000,C 90.000,E1 274.702} C_DIS
LIN {X -0.140,Y -342.774,Z 1817.523,A 0.000,B 0.000,C 90.000,E1 274.131} C_DIS
LIN {X -0.035,Y -336.869,Z 1817.520,A 0.000,B 0.000,C 90.000,E1 273.555} C_DIS
LIN {X -0.021,Y -330.716,Z 1817.517,A 0.000,B 0.000,C 90.000,E1 273.037} C_DIS
LIN {X -0.089,Y -324.405,Z 1817.514,A 0.000,B 0.000,C 90.000,E1 272.579} C_DIS
LIN {X 0.104,Y -317.868,Z 1817.512,A 0.000,B 0.000,C 90.000,E1 272.121} C_DIS
LIN {X -0.064,Y -311.024,Z 1817.510,A 0.000,B 0.000,C 90.000,E1 271.776} C_DIS
LIN {X 0.058,Y -303.780,Z 1817.508,A 0.000,B 0.000,C 90.000,E1 271.432} C_DIS
LIN {X -0.132,Y -296.394,Z 1817.507,A 0.000,B 0.000,C 90.000,E1 271.203} C_DIS
LIN {X -0.048,Y -288.764,Z 1817.505,A 0.000,B 0.000,C 90.000,E1 270.974} C_DIS
LIN {X 0.096,Y -273.847,Z 1817.504,A 0.000,B 0.000,C 90.000,E1 270.630} C_DIS
LIN {X 0.100,Y -251.736,Z 1817.501,A 0.000,B 0.000,C 90.000,E1 270.229} C_DIS
LIN {X 0.084,Y -241.665,Z 1817.501,A 0.000,B 0.000,C 90.000,E1 270.115} C_DIS
LIN {X -0.113,Y -232.389,Z 1817.500,A 0.000,B 0.000,C 90.000,E1 270.115} C_DIS
LIN {X 0.068,Y -181.571,Z 1817.500,A 0.000,B 0.000,C 90.000,E1 270.057} C_DIS
LIN {X -0.004,Y -180.907,Z 1817.475,A 0.000,B 0.000,C 90.000,E1 265.527} C_DIS
LIN {X 0.053,Y -180.761,Z 1817.470,A 0.000,B 0.000,C 90.000,E1 264.666} C_DIS
LIN {X -0.055,Y -178.854,Z 1817.442,A 0.000,B 0.000,C 90.000,E1 259.634} C_DIS
LIN {X 0.017,Y -175.897,Z 1817.414,A 0.000,B 0.000,C 90.000,E1 254.519} C_DIS
LIN {X -0.044,Y -174.574,Z 1817.405,A 0.000,B 0.000,C 90.000,E1 252.834} C_DIS
LIN {X -0.008,Y -171.557,Z 1817.381,A 0.000,B 0.000,C 90.000,E1 248.539} C_DIS
LIN {X 0.047,Y -167.781,Z 1817.357,A 0.000,B 0.000,C 90.000,E1 244.204} C_DIS
LIN {X -0.012,Y -166.493,Z 1817.347,A 0.000,B 0.000,C 90.000,E1 242.487} C_DIS
LIN {X -0.016,Y -163.203,Z 1817.328,A 0.000,B 0.000,C 90.000,E1 238.997} C_DIS
LIN {X 0.039,Y -161.168,Z 1817.313,A 0.000,B 0.000,C 90.000,E1 236.342} C_DIS
LIN {X 0.073,Y -157.182,Z 1817.288,A 0.000,B 0.000,C 90.000,E1 231.904} C_DIS
LIN {X -0.004,Y -155.913,Z 1817.279,A 0.000,B 0.000,C 90.000,E1 230.150} C_DIS
LIN {X 0.053,Y -152.163,Z 1817.254,A 0.000,B 0.000,C 90.000,E1 225.648} C_DIS
LIN {X 0.073,Y -150.412,Z 1817.239,A 0.000,B 0.000,C 90.000,E1 222.933} C_DIS
LIN {X 0.004,Y -147.141,Z 1817.214,A 0.000,B 0.000,C 90.000,E1 218.418} C_DIS
LIN {X 0.002,Y -145.700,Z 1817.198,A 0.000,B 0.000,C 90.000,E1 215.678} C_DIS
LIN {X 0.009,Y -143.083,Z 1817.173,A 0.000,B 0.000,C 90.000,E1 211.082} C_DIS
LIN {X 0.014,Y -141.701,Z 1817.152,A 0.000,B 0.000,C 90.000,E1 207.385} C_DIS
LIN {X -0.064,Y -139.466,Z 1817.116,A 0.000,B 0.000,C 90.000,E1 200.918} C_DIS
LIN {X -0.010,Y -139.200,Z 1817.106,A 0.000,B 0.000,C 90.000,E1 199.033} C_DIS
LIN {X 0.054,Y -138.327,Z 1817.054,A 0.000,B 0.000,C 90.000,E1 189.670} C_DIS
LIN {X 0.059,Y -139.445,Z 1817.007,A 0.000,B 0.000,C 90.000,E1 181.260} C_DIS
LIN {X 0.000,Y -140.983,Z 1816.976,A 0.000,B 0.000,C 90.000,E1 175.698} C_DIS
LIN {X -0.051,Y -142.739,Z 1816.955,A 0.000,B 0.000,C 90.000,E1 172.008} C_DIS
LIN {X 0.047,Y -145.131,Z 1816.930,A 0.000,B 0.000,C 90.000,E1 167.353} C_DIS
LIN {X 0.041,Y -147.754,Z 1816.909,A 0.000,B 0.000,C 90.000,E1 163.685} C_DIS
LIN {X -0.020,Y -150.424,Z 1816.889,A 0.000,B 0.000,C 90.000,E1 160.061} C_DIS
LIN {X -0.005,Y -153.865,Z 1816.869,A 0.000,B 0.000,C 90.000,E1 156.433} C_DIS
LIN {X -0.088,Y -157.276,Z 1816.849,A 0.000,B 0.000,C 90.000,E1 152.871} C_DIS
LIN {X -0.011,Y -161.454,Z 1816.829,A 0.000,B 0.000,C 90.000,E1 149.282} C_DIS
LIN {X -0.004,Y -165.655,Z 1816.810,A 0.000,B 0.000,C 90.000,E1 145.754} C_DIS
LIN {X -0.022,Y -170.590,Z 1816.790,A 0.000,B 0.000,C 90.000,E1 142.271} C_DIS
LIN {X 0.017,Y -175.468,Z 1816.771,A 0.000,B 0.000,C 90.000,E1 138.809} C_DIS
LIN {X -0.001,Y -181.090,Z 1816.752,A 0.000,B 0.000,C 90.000,E1 135.405} C_DIS
LIN {X -0.011,Y -186.532,Z 1816.734,A 0.000,B 0.000,C 90.000,E1 132.043} C_DIS
LIN {X -0.069,Y -191.149,Z 1816.720,A 0.000,B 0.000,C 90.000,E1 129.564} C_DIS
LIN {X 0.009,Y -196.950,Z 1816.701,A 0.000,B 0.000,C 90.000,E1 126.251} C_DIS
LIN {X 0.045,Y -200.215,Z 1816.692,A 0.000,B 0.000,C 90.000,E1 124.612} C_DIS
LIN {X 0.040,Y -207.709,Z 1816.670,A 0.000,B 0.000,C 90.000,E1 120.590} C_DIS
LIN {X 0.043,Y -210.892,Z 1816.661,A 0.000,B 0.000,C 90.000,E1 118.999} C_DIS
LIN {X 0.050,Y -216.756,Z 1816.644,A 0.000,B 0.000,C 90.000,E1 115.848} C_DIS
LIN {X -0.131,Y -219.813,Z 1816.635,A 0.000,B 0.000,C 90.000,E1 114.335} C_DIS
LIN {X -0.014,Y -224.018,Z 1816.622,A 0.000,B 0.000,C 90.000,E1 111.897} C_DIS
LIN {X -0.052,Y -283.578,Z 1816.622,A 0.000,B 0.000,C 90.000,E1 111.897} C_DIS
LIN {X -0.162,Y -286.534,Z 1816.621,A 0.000,B 0.000,C 90.000,E1 111.844} C_DIS
LIN {X -0.125,Y -291.142,Z 1816.620,A 0.000,B 0.000,C 90.000,E1 111.535} C_DIS
LIN {X -0.086,Y -293.848,Z 1816.618,A 0.000,B 0.000,C 90.000,E1 111.227} C_DIS
LIN {X -0.091,Y -295.896,Z 1816.616,A 0.000,B 0.000,C 90.000,E1 110.918} C_DIS
LIN {X 0.033,Y -308.956,Z 1816.603,A 0.000,B 0.000,C 90.000,E1 108.598} C_DIS
LIN {X 0.127,Y -323.490,Z 1816.591,A 0.000,B 0.000,C 90.000,E1 106.315} C_DIS
LIN {X 0.088,Y -337.130,Z 1816.580,A 0.000,B 0.000,C 90.000,E1 104.426} C_DIS
LIN {X -0.020,Y -351.953,Z 1816.570,A 0.000,B 0.000,C 90.000,E1 102.591} C_DIS
LIN {X -0.042,Y -370.340,Z 1816.559,A 0.000,B 0.000,C 90.000,E1 100.546} C_DIS
LIN {X -0.005,Y -389.153,Z 1816.548,A 0.000,B 0.000,C 90.000,E1 98.681} C_DIS
LIN {X -0.143,Y -408.385,Z 1816.539,A 0.000,B 0.000,C 90.000,E1 97.004} C_DIS
LIN {X 0.057,Y -430.745,Z 1816.529,A 0.000,B 0.000,C 90.000,E1 95.220} C_DIS
LIN {X 0.212,Y -439.149,Z 1816.526,A 0.000,B 0.000,C 90.000,E1 94.588} C_DIS
LIN {X -0.014,Y -441.310,Z 1816.525,A 0.000,B 0.000,C 90.000,E1 94.416} C_DIS
LIN {X -0.117,Y -443.280,Z 1816.523,A 0.000,B 0.000,C 90.000,E1 94.188} C_DIS
LIN {X -0.190,Y -444.789,Z 1816.522,A 0.000,B 0.000,C 90.000,E1 93.955} C_DIS
LIN {X -0.012,Y -446.044,Z 1816.520,A 0.000,B 0.000,C 90.000,E1 93.669} C_DIS
LIN {X 0.168,Y -446.973,Z 1816.519,A 0.000,B 0.000,C 90.000,E1 93.383} C_DIS
LIN {X 0.124,Y -448.018,Z 1816.516,A 0.000,B 0.000,C 90.000,E1 92.865} C_DIS
LIN {X 0.063,Y -448.112,Z 1816.513,A 0.000,B 0.000,C 90.000,E1 92.350} C_DIS
LIN {X 0.010,Y -447.273,Z 1816.510,A 0.000,B 0.000,C 90.000,E1 91.835} C_DIS
LIN {X -0.030,Y -445.366,Z 1816.507,A 0.000,B 0.000,C 90.000,E1 91.318} C_DIS
LIN {X -0.085,Y -442.242,Z 1816.504,A 0.000,B 0.000,C 90.000,E1 90.802} C_DIS
LIN {X -0.057,Y -429.053,Z 1816.493,A 0.000,B 0.000,C 90.000,E1 88.682} C_DIS
LIN {X 0.005,Y -417.294,Z 1816.482,A 0.000,B 0.000,C 90.000,E1 86.788} C_DIS
LIN {X 0.174,Y -407.164,Z 1816.473,A 0.000,B 0.000,C 90.000,E1 85.122} C_DIS
LIN {X -0.168,Y -395.255,Z 1816.462,A 0.000,B 0.000,C 90.000,E1 83.223} C_DIS
LIN {X 0.115,Y -383.301,Z 1816.451,A 0.000,B 0.000,C 90.000,E1 81.197} C_DIS
LIN {X 0.200,Y -369.695,Z 1816.438,A 0.000,B 0.000,C 90.000,E1 78.870} C_DIS
LIN {X -0.037,Y -351.914,Z 1816.420,A 0.000,B 0.000,C 90.000,E1 75.644} C_DIS
LIN {X -0.047,Y -338.220,Z 1816.405,A 0.000,B 0.000,C 90.000,E1 72.906} C_DIS
LIN {X -0.047,Y -327.838,Z 1816.393,A 0.000,B 0.000,C 90.000,E1 70.732} C_DIS
LIN {X 0.055,Y -313.461,Z 1816.375,A 0.000,B 0.000,C 90.000,E1 67.539} C_DIS
LIN {X -0.009,Y -303.815,Z 1816.363,A 0.000,B 0.000,C 90.000,E1 65.281} C_DIS
LIN {X -0.152,Y -292.662,Z 1816.348,A 0.000,B 0.000,C 90.000,E1 62.615} C_DIS
LIN {X 0.053,Y -292.638,Z 1816.348,A 0.000,B 0.000,C 90.000,E1 62.564} C_DIS
LIN {X -0.040,Y -298.614,Z 1816.339,A 0.000,B 0.000,C 90.000,E1 60.973} C_DIS
LIN {X -0.171,Y -300.085,Z 1816.335,A 0.000,B 0.000,C 90.000,E1 60.333} C_DIS
LIN {X -0.146,Y -299.804,Z 1816.331,A 0.000,B 0.000,C 90.000,E1 59.665} C_DIS
LIN {X -0.111,Y -298.901,Z 1816.328,A 0.000,B 0.000,C 90.000,E1 58.997} C_DIS
LIN {X -0.077,Y -297.637,Z 1816.324,A 0.000,B 0.000,C 90.000,E1 58.329} C_DIS
LIN {X -0.035,Y -294.513,Z 1816.317,A 0.000,B 0.000,C 90.000,E1 56.993} C_DIS
LIN {X -0.117,Y -290.936,Z 1816.309,A 0.000,B 0.000,C 90.000,E1 55.674} C_DIS
LIN {X 0.050,Y -284.968,Z 1816.298,A 0.000,B 0.000,C 90.000,E1 53.623} C_DIS
LIN {X -0.122,Y -278.652,Z 1816.287,A 0.000,B 0.000,C 90.000,E1 51.618} C_DIS
LIN {X -0.067,Y -272.217,Z 1816.275,A 0.000,B 0.000,C 90.000,E1 49.542} C_DIS
LIN {X -0.037,Y -263.609,Z 1816.260,A 0.000,B 0.000,C 90.000,E1 46.743} C_DIS
LIN {X 0.069,Y -257.192,Z 1816.248,A 0.000,B 0.000,C 90.000,E1 44.595} C_DIS
LIN {X 0.051,Y -250.804,Z 1816.236,A 0.000,B 0.000,C 90.000,E1 42.447} C_DIS
LIN {X -0.071,Y -244.382,Z 1816.224,A 0.000,B 0.000,C 90.000,E1 40.297} C_DIS
LIN {X 0.059,Y -235.836,Z 1816.207,A 0.000,B 0.000,C 90.000,E1 37.317} C_DIS
LIN {X 0.021,Y -227.381,Z 1816.191,A 0.000,B 0.000,C 90.000,E1 34.326} C_DIS
LIN {X 0.077,Y -219.535,Z 1816.174,A 0.000,B 0.000,C 90.000,E1 31.258} C_DIS
LIN {X 0.083,Y -212.228,Z 1816.156,A 0.000,B 0.000,C 90.000,E1 28.153} C_DIS
LIN {X -0.010,Y -205.600,Z 1816.139,A 0.000,B 0.000,C 90.000,E1 25.027} C_DIS
LIN {X -0.036,Y -201.147,Z 1816.126,A 0.000,B 0.000,C 90.000,E1 22.642} C_DIS
LIN {X 0.032,Y -196.119,Z 1816.108,A 0.000,B 0.000,C 90.000,E1 19.396} C_DIS
LIN {X 0.030,Y -191.912,Z 1816.090,A 0.000,B 0.000,C 90.000,E1 16.134} C_DIS
LIN {X 0.057,Y -187.690,Z 1816.067,A 0.000,B 0.000,C 90.000,E1 12.007} C_DIS
LIN {X -0.010,Y -184.500,Z 1816.044,A 0.000,B 0.000,C 90.000,E1 7.871} C_DIS
LIN {X -0.012,Y -181.632,Z 1816.011,A 0.000,B 0.000,C 90.000,E1 2.007} C_DIS
LIN {X -0.053,Y -180.508,Z 1815.969,A 0.000,B 0.000,C 90.000,E1 354.489} C_DIS
LIN {X 0.075,Y -181.404,Z 1815.932,A 0.000,B 0.000,C 90.000,E1 347.701} C_DIS
LIN {X 0.061,Y -183.453,Z 1815.899,A 0.000,B 0.000,C 90.000,E1 341.819} C_DIS
LIN {X 0.075,Y -186.283,Z 1815.871,A 0.000,B 0.000,C 90.000,E1 336.794} C_DIS
LIN {X -0.023,Y -189.211,Z 1815.848,A 0.000,B 0.000,C 90.000,E1 332.666} C_DIS
LIN {X -0.006,Y -193.496,Z 1815.821,A 0.000,B 0.000,C 90.000,E1 327.709} C_DIS
LIN {X -0.015,Y -197.752,Z 1815.798,A 0.000,B 0.000,C 90.000,E1 323.623} C_DIS
LIN {X 0.072,Y -201.931,Z 1815.780,A 0.000,B 0.000,C 90.000,E1 320.356} C_DIS
LIN {X 0.023,Y -205.780,Z 1815.766,A 0.000,B 0.000,C 90.000,E1 317.957} C_DIS
LIN {X -0.038,Y -208.797,Z 1815.758,A 0.000,B 0.000,C 90.000,E1 316.377} C_DIS
LIN {X 0.085,Y -212.264,Z 1815.749,A 0.000,B 0.000,C 90.000,E1 314.757} C_DIS
LIN {X 0.004,Y -217.391,Z 1815.738,A 0.000,B 0.000,C 90.000,E1 312.813} C_DIS
LIN {X 0.114,Y -222.213,Z 1815.729,A 0.000,B 0.000,C 90.000,E1 311.229} C_DIS
LIN {X -0.023,Y -227.846,Z 1815.721,A 0.000,B 0.000,C 90.000,E1 309.725} C_DIS
LIN {X 0.086,Y -234.222,Z 1815.712,A 0.000,B 0.000,C 90.000,E1 308.177} C_DIS
LIN {X 0.111,Y -243.077,Z 1815.702,A 0.000,B 0.000,C 90.000,E1 306.297} C_DIS
LIN {X 0.000,Y -254.951,Z 1815.690,A 0.000,B 0.000,C 90.000,E1 304.119} C_DIS
LIN {X 0.048,Y -267.891,Z 1815.678,A 0.000,B 0.000,C 90.000,E1 301.957} C_DIS
LIN {X 0.104,Y -289.284,Z 1815.660,A 0.000,B 0.000,C 90.000,E1 298.821} C_DIS
LIN {X 0.025,Y -304.087,Z 1815.649,A 0.000,B 0.000,C 90.000,E1 296.821} C_DIS
LIN {X 0.095,Y -319.347,Z 1815.638,A 0.000,B 0.000,C 90.000,E1 294.847} C_DIS
LIN {X 0.057,Y -331.993,Z 1815.629,A 0.000,B 0.000,C 90.000,E1 293.259} C_DIS
LIN {X -0.045,Y -341.850,Z 1815.622,A 0.000,B 0.000,C 90.000,E1 292.025} C_DIS
LIN {X -0.023,Y -351.359,Z 1815.615,A 0.000,B 0.000,C 90.000,E1 290.791} C_DIS
LIN {X -0.050,Y -358.103,Z 1815.610,A 0.000,B 0.000,C 90.000,E1 289.885} C_DIS
LIN {X 0.104,Y -364.225,Z 1815.605,A 0.000,B 0.000,C 90.000,E1 288.960} C_DIS
LIN {X 0.204,Y -369.688,Z 1815.600,A 0.000,B 0.000,C 90.000,E1 288.055} C_DIS
LIN {X -0.116,Y -374.355,Z 1815.596,A 0.000,B 0.000,C 90.000,E1 287.221} C_DIS
LIN {X 0.078,Y -378.104,Z 1815.591,A 0.000,B 0.000,C 90.000,E1 286.315} C_DIS
LIN {X 0.200,Y -381.046,Z 1815.586,A 0.000,B 0.000,C 90.000,E1 285.426} C_DIS
LIN {X -0.142,Y -382.576,Z 1815.583,A 0.000,B 0.000,C 90.000,E1 284.898} C_DIS
LIN {X -0.005,Y -383.717,Z 1815.579,A 0.000,B 0.000,C 90.000,E1 284.300} C_DIS
LIN {X 0.049,Y -384.451,Z 1815.576,A 0.000,B 0.000,C 90.000,E1 283.716} C_DIS
LIN {X 0.200,Y -384.777,Z 1815.573,A 0.000,B 0.000,C 90.000,E1 283.119} C_DIS
LIN {X -0.109,Y -384.727,Z 1815.570,A 0.000,B 0.000,C 90.000,E1 282.591} C_DIS
LIN {X -0.039,Y -384.170,Z 1815.567,A 0.000,B 0.000,C 90.000,E1 282.007} C_DIS
LIN {X 0.031,Y -383.247,Z 1815.563,A 0.000,B 0.000,C 90.000,E1 281.422} C_DIS
LIN {X 0.097,Y -381.890,Z 1815.560,A 0.000,B 0.000,C 90.000,E1 280.838} C_DIS
LIN {X 0.156,Y -380.193,Z 1815.557,A 0.000,B 0.000,C 90.000,E1 280.254} C_DIS
LIN {X -0.148,Y -377.065,Z 1815.552,A 0.000,B 0.000,C 90.000,E1 279.434} C_DIS
LIN {X -0.169,Y -373.363,Z 1815.547,A 0.000,B 0.000,C 90.000,E1 278.568} C_DIS
LIN {X 0.141,Y -369.151,Z 1815.543,A 0.000,B 0.000,C 90.000,E1 277.644} C_DIS
LIN {X 0.050,Y -364.242,Z 1815.538,A 0.000,B 0.000,C 90.000,E1 276.777} C_DIS
LIN {X -0.048,Y -360.462,Z 1815.534,A 0.000,B 0.000,C 90.000,E1 276.201} C_DIS
LIN {X -0.165,Y -356.212,Z 1815.531,A 0.000,B 0.000,C 90.000,E1 275.625} C_DIS
LIN {X 0.048,Y -351.393,Z 1815.528,A 0.000,B 0.000,C 90.000,E1 274.992} C_DIS
LIN {X -0.032,Y -346.002,Z 1815.525,A 0.000,B 0.000,C 90.000,E1 274.416} C_DIS
LIN {X -0.026,Y -340.254,Z 1815.521,A 0.000,B 0.000,C 90.000,E1 273.841} C_DIS
LIN {X -0.174,Y -334.178,Z 1815.518,A 0.000,B 0.000,C 90.000,E1 273.326} C_DIS
LIN {X -0.042,Y -327.841,Z 1815.516,A 0.000,B 0.000,C 90.000,E1 272.808} C_DIS
LIN {X 0.027,Y -321.475,Z 1815.513,A 0.000,B 0.000,C 90.000,E1 272.350} C_DIS
LIN {X -0.029,Y -314.587,Z 1815.511,A 0.000,B 0.000,C 90.000,E1 271.949} C_DIS
LIN {X -0.042,Y -307.683,Z 1815.509,A 0.000,B 0.000,C 90.000,E1 271.604} C_DIS
LIN {X -0.103,Y -300.154,Z 1815.507,A 0.000,B 0.000,C 90.000,E1 271.318} C_DIS
LIN {X 0.140,Y -292.480,Z 1815.506,A 0.000,B 0.000,C 90.000,E1 271.031} C_DIS
LIN {X -0.032,Y -281.102,Z 1815.504,A 0.000,B 0.000,C 90.000,E1 270.802} C_DIS
LIN {X -0.060,Y -262.526,Z 1815.502,A 0.000,B 0.000,C 90.000,E1 270.458} C_DIS
LIN {X 0.093,Y -251.369,Z 1815.501,A 0.000,B 0.000,C 90.000,E1 270.229} C_DIS
LIN {X 0.080,Y -240.737,Z 1815.501,A 0.000,B 0.000,C 90.000,E1 270.115} C_DIS
LIN {X -0.077,Y -233.300,Z 1815.500,A 0.000,B 0.000,C 90.000,E1 270.115} C_DIS
LIN {X -0.083,Y -181.572,Z 1815.500,A 0.000,B 0.000,C 90.000,E1 270.115} C_DIS
LIN {X 0.004,Y -180.908,Z 1815.475,A 0.000,B 0.000,C 90.000,E1 265.527} C_DIS
LIN {X 0.060,Y -180.761,Z 1815.470,A 0.000,B 0.000,C 90.000,E1 264.666} C_DIS
LIN {X -0.047,Y -178.855,Z 1815.442,A 0.000,B 0.000,C 90.000,E1 259.634} C_DIS
LIN {X 0.024,Y -175.899,Z 1815.414,A 0.000,B 0.000,C 90.000,E1 254.519} C_DIS
LIN {X -0.037,Y -174.576,Z 1815.405,A 0.000,B 0.000,C 90.000,E1 252.834} C_DIS
LIN {X -0.002,Y -171.559,Z 1815.381,A 0.000,B 0.000,C 90.000,E1 248.539} C_DIS
LIN {X 0.054,Y -167.782,Z 1815.357,A 0.000,B 0.000,C 90.000,E1 244.204} C_DIS
LIN {X -0.005,Y -166.496,Z 1815.347,A 0.000,B 0.000,C 90.000,E1 242.487} C_DIS
LIN {X -0.009,Y -163.205,Z 1815.328,A 0.000,B 0.000,C 90.000,E1 238.997} C_DIS
LIN {X -0.044,Y -161.170,Z 1815.313,A 0.000,B 0.000,C 90.000,E1 236.373} C_DIS
LIN {X 0.080,Y -157.184,Z 1815.289,A 0.000,B 0.000,C 90.000,E1 231.904} C_DIS
LIN {X 0.003,Y -155.915,Z 1815.279,A 0.000,B 0.000,C 90.000,E1 230.150} C_DIS
LIN {X 0.060,Y -152.165,Z 1815.254,A 0.000,B 0.000,C 90.000,E1 225.648} C_DIS
LIN {X -0.032,Y -150.413,Z 1815.239,A 0.000,B 0.000,C 90.000,E1 222.975} C_DIS
LIN {X 0.010,Y -147.142,Z 1815.214,A 0.000,B 0.000,C 90.000,E1 218.418} C_DIS
LIN {X 0.007,Y -145.701,Z 1815.198,A 0.000,B 0.000,C 90.000,E1 215.678} C_DIS
LIN {X 0.015,Y -143.084,Z 1815.173,A 0.000,B 0.000,C 90.000,E1 211.082} C_DIS
LIN {X 0.020,Y -141.702,Z 1815.152,A 0.000,B 0.000,C 90.000,E1 207.385} C_DIS
LIN {X -0.057,Y -139.467,Z 1815.116,A 0.000,B 0.000,C 90.000,E1 200.918} C_DIS
LIN {X -0.003,Y -139.200,Z 1815.106,A 0.000,B 0.000,C 90.000,E1 199.033} C_DIS
LIN {X 0.060,Y -138.327,Z 1815.054,A 0.000,B 0.000,C 90.000,E1 189.670} C_DIS
LIN {X 0.065,Y -139.444,Z 1815.007,A 0.000,B 0.000,C 90.000,E1 181.260} C_DIS
LIN {X 0.006,Y -140.983,Z 1814.976,A 0.000,B 0.000,C 90.000,E1 175.698} C_DIS
LIN {X -0.045,Y -142.738,Z 1814.955,A 0.000,B 0.000,C 90.000,E1 172.008} C_DIS
LIN {X 0.054,Y -145.129,Z 1814.930,A 0.000,B 0.000,C 90.000,E1 167.353} C_DIS
LIN {X 0.048,Y -147.752,Z 1814.909,A 0.000,B 0.000,C 90.000,E1 163.685} C_DIS
LIN {X -0.013,Y -150.421,Z 1814.889,A 0.000,B 0.000,C 90.000,E1 160.061} C_DIS
LIN {X 0.002,Y -153.863,Z 1814.869,A 0.000,B 0.000,C 90.000,E1 156.433} C_DIS
LIN {X -0.082,Y -157.273,Z 1814.849,A 0.000,B 0.000,C 90.000,E1 152.871} C_DIS
LIN {X -0.005,Y -161.452,Z 1814.829,A 0.000,B 0.000,C 90.000,E1 149.282} C_DIS
LIN {X 0.003,Y -165.652,Z 1814.810,A 0.000,B 0.000,C 90.000,E1 145.754} C_DIS
LIN {X -0.016,Y -170.587,Z 1814.790,A 0.000,B 0.000,C 90.000,E1 142.271} C_DIS
LIN {X -0.109,Y -175.464,Z 1814.771,A 0.000,B 0.000,C 90.000,E1 138.852} C_DIS
LIN {X 0.006,Y -181.086,Z 1814.752,A 0.000,B 0.000,C 90.000,E1 135.405} C_DIS
LIN {X -0.003,Y -186.528,Z 1814.734,A 0.000,B 0.000,C 90.000,E1 132.043} C_DIS
LIN {X -0.062,Y -191.145,Z 1814.720,A 0.000,B 0.000,C 90.000,E1 129.564} C_DIS
LIN {X 0.016,Y -196.946,Z 1814.701,A 0.000,B 0.000,C 90.000,E1 126.251} C_DIS
LIN {X 0.052,Y -200.210,Z 1814.692,A 0.000,B 0.000,C 90.000,E1 124.612} C_DIS
LIN {X 0.048,Y -207.704,Z 1814.670,A 0.000,B 0.000,C 90.000,E1 120.590} C_DIS
LIN {X 0.051,Y -210.889,Z 1814.661,A 0.000,B 0.000,C 90.000,E1 118.999} C_DIS
LIN {X 0.058,Y -216.752,Z 1814.644,A 0.000,B 0.000,C 90.000,E1 115.848} C_DIS
LIN {X -0.123,Y -219.809,Z 1814.635,A 0.000,B 0.000,C 90.000,E1 114.335} C_DIS
LIN {X -0.006,Y -224.014,Z 1814.622,A 0.000,B 0.000,C 90.000,E1 111.897} C_DIS
LIN {X -0.042,Y -283.540,Z 1814.622,A 0.000,B 0.000,C 90.000,E1 111.897} C_DIS
LIN {X -0.152,Y -286.515,Z 1814.621,A 0.000,B 0.000,C 90.000,E1 111.844} C_DIS
LIN {X -0.115,Y -291.128,Z 1814.620,A 0.000,B 0.000,C 90.000,E1 111.535} C_DIS
LIN {X -0.076,Y -293.835,Z 1814.618,A 0.000,B 0.000,C 90.000,E1 111.227} C_DIS
LIN {X -0.081,Y -295.882,Z 1814.616,A 0.000,B 0.000,C 90.000,E1 110.918} C_DIS
LIN {X 0.045,Y -308.942,Z 1814.603,A 0.000,B 0.000,C 90.000,E1 108.598} C_DIS
LIN {X 0.139,Y -323.474,Z 1814.591,A 0.000,B 0.000,C 90.000,E1 106.315} C_DIS
LIN {X 0.100,Y -337.113,Z 1814.580,A 0.000,B 0.000,C 90.000,E1 104.426} C_DIS
LIN {X -0.008,Y -351.934,Z 1814.570,A 0.000,B 0.000,C 90.000,E1 102.591} C_DIS
LIN {X -0.031,Y -370.320,Z 1814.559,A 0.000,B 0.000,C 90.000,E1 100.546} C_DIS
LIN {X 0.006,Y -389.135,Z 1814.548,A 0.000,B 0.000,C 90.000,E1 98.681} C_DIS
LIN {X -0.133,Y -408.366,Z 1814.539,A 0.000,B 0.000,C 90.000,E1 97.004} C_DIS
LIN {X 0.067,Y -430.726,Z 1814.529,A 0.000,B 0.000,C 90.000,E1 95.220} C_DIS
LIN {X 0.221,Y -439.131,Z 1814.526,A 0.000,B 0.000,C 90.000,E1 94.588} C_DIS
LIN {X -0.005,Y -441.293,Z 1814.525,A 0.000,B 0.000,C 90.000,E1 94.416} C_DIS
LIN {X -0.107,Y -443.263,Z 1814.523,A 0.000,B 0.000,C 90.000,E1 94.188} C_DIS
LIN {X -0.180,Y -444.773,Z 1814.522,A 0.000,B 0.000,C 90.000,E1 93.955} C_DIS
LIN {X -0.001,Y -446.027,Z 1814.520,A 0.000,B 0.000,C 90.000,E1 93.669} C_DIS
LIN {X 0.178,Y -446.958,Z 1814.519,A 0.000,B 0.000,C 90.000,E1 93.383} C_DIS
LIN {X 0.135,Y -448.005,Z 1814.516,A 0.000,B 0.000,C 90.000,E1 92.865} C_DIS
LIN {X 0.073,Y -448.100,Z 1814.513,A 0.000,B 0.000,C 90.000,E1 92.350} C_DIS
LIN {X 0.020,Y -447.260,Z 1814.510,A 0.000,B 0.000,C 90.000,E1 91.835} C_DIS
LIN {X -0.019,Y -445.356,Z 1814.507,A 0.000,B 0.000,C 90.000,E1 91.318} C_DIS
LIN {X -0.076,Y -442.232,Z 1814.504,A 0.000,B 0.000,C 90.000,E1 90.802} C_DIS
LIN {X -0.048,Y -429.043,Z 1814.493,A 0.000,B 0.000,C 90.000,E1 88.682} C_DIS
LIN {X 0.014,Y -417.284,Z 1814.482,A 0.000,B 0.000,C 90.000,E1 86.788} C_DIS
LIN {X 0.183,Y -407.152,Z 1814.473,A 0.000,B 0.000,C 90.000,E1 85.122} C_DIS
LIN {X -0.161,Y -395.244,Z 1814.462,A 0.000,B 0.000,C 90.000,E1 83.223} C_DIS
LIN {X 0.122,Y -383.291,Z 1814.451,A 0.000,B 0.000,C 90.000,E1 81.197} C_DIS
LIN {X -0.156,Y -369.683,Z 1814.438,A 0.000,B 0.000,C 90.000,E1 78.926} C_DIS
LIN {X -0.031,Y -351.901,Z 1814.420,A 0.000,B 0.000,C 90.000,E1 75.644} C_DIS
LIN {X -0.041,Y -338.205,Z 1814.405,A 0.000,B 0.000,C 90.000,E1 72.906} C_DIS
LIN {X -0.042,Y -327.823,Z 1814.393,A 0.000,B 0.000,C 90.000,E1 70.732} C_DIS
LIN {X 0.060,Y -313.444,Z 1814.375,A 0.000,B 0.000,C 90.000,E1 67.539} C_DIS
LIN {X -0.005,Y -303.796,Z 1814.363,A 0.000,B 0.000,C 90.000,E1 65.281} C_DIS
LIN {X -0.161,Y -300.005,Z 1814.358,A 0.000,B 0.000,C 90.000,E1 64.409} C_DIS
LIN {X 0.056,Y -299.968,Z 1814.358,A 0.000,B 0.000,C 90.000,E1 64.357} C_DIS
LIN {X 0.045,Y -307.213,Z 1814.346,A 0.000,B 0.000,C 90.000,E1 62.308} C_DIS
LIN {X 0.114,Y -307.625,Z 1814.343,A 0.000,B 0.000,C 90.000,E1 61.641} C_DIS
LIN {X 0.042,Y -307.039,Z 1814.339,A 0.000,B 0.000,C 90.000,E1 61.001} C_DIS
LIN {X 0.122,Y -305.966,Z 1814.335,A 0.000,B 0.000,C 90.000,E1 60.333} C_DIS
LIN {X -0.064,Y -304.606,Z 1814.332,A 0.000,B 0.000,C 90.000,E1 59.715} C_DIS
LIN {X -0.083,Y -301.340,Z 1814.324,A 0.000,B 0.000,C 90.000,E1 58.408} C_DIS
LIN {X 0.169,Y -297.561,Z 1814.317,A 0.000,B 0.000,C 90.000,E1 57.041} C_DIS
LIN {X -0.114,Y -291.430,Z 1814.306,A 0.000,B 0.000,C 90.000,E1 55.102} C_DIS
LIN {X 0.032,Y -283.754,Z 1814.293,A 0.000,B 0.000,C 90.000,E1 52.718} C_DIS
LIN {X -0.116,Y -275.837,Z 1814.280,A 0.000,B 0.000,C 90.000,E1 50.356} C_DIS
LIN {X -0.081,Y -267.927,Z 1814.266,A 0.000,B 0.000,C 90.000,E1 47.919} C_DIS
LIN {X -0.004,Y -259.005,Z 1814.250,A 0.000,B 0.000,C 90.000,E1 45.081} C_DIS
LIN {X -0.165,Y -251.244,Z 1814.236,A 0.000,B 0.000,C 90.000,E1 42.609} C_DIS
LIN {X 0.050,Y -243.439,Z 1814.222,A 0.000,B 0.000,C 90.000,E1 40.011} C_DIS
LIN {X 0.106,Y -233.588,Z 1814.204,A 0.000,B 0.000,C 90.000,E1 36.664} C_DIS
LIN {X 0.068,Y -225.262,Z 1814.187,A 0.000,B 0.000,C 90.000,E1 33.658} C_DIS
LIN {X 0.072,Y -217.468,Z 1814.170,A 0.000,B 0.000,C 90.000,E1 30.590} C_DIS
LIN {X -0.074,Y -210.302,Z 1814.153,A 0.000,B 0.000,C 90.000,E1 27.513} C_DIS
LIN {X -0.020,Y -203.855,Z 1814.135,A 0.000,B 0.000,C 90.000,E1 24.335} C_DIS
LIN {X 0.105,Y -199.544,Z 1814.122,A 0.000,B 0.000,C 90.000,E1 21.897} C_DIS
LIN {X 0.064,Y -194.701,Z 1814.104,A 0.000,B 0.000,C 90.000,E1 18.671} C_DIS
LIN {X -0.028,Y -190.633,Z 1814.086,A 0.000,B 0.000,C 90.000,E1 15.426} C_DIS
LIN {X -0.037,Y -186.627,Z 1814.063,A 0.000,B 0.000,C 90.000,E1 11.299} C_DIS
LIN {X 0.084,Y -183.160,Z 1814.035,A 0.000,B 0.000,C 90.000,E1 6.258} C_DIS
LIN {X -0.032,Y -180.577,Z 1813.997,A 0.000,B 0.000,C 90.000,E1 359.542} C_DIS
LIN {X -0.015,Y -180.133,Z 1813.965,A 0.000,B 0.000,C 90.000,E1 353.628} C_DIS
LIN {X -0.031,Y -181.243,Z 1813.927,A 0.000,B 0.000,C 90.000,E1 346.881} C_DIS
LIN {X 0.052,Y -183.518,Z 1813.894,A 0.000,B 0.000,C 90.000,E1 340.967} C_DIS
LIN {X -0.032,Y -186.526,Z 1813.866,A 0.000,B 0.000,C 90.000,E1 335.973} C_DIS
LIN {X -0.037,Y -189.580,Z 1813.843,A 0.000,B 0.000,C 90.000,E1 331.820} C_DIS
LIN {X 0.074,Y -193.236,Z 1813.820,A 0.000,B 0.000,C 90.000,E1 327.661} C_DIS
LIN {X 0.050,Y -197.566,Z 1813.798,A 0.000,B 0.000,C 90.000,E1 323.577} C_DIS
LIN {X -0.029,Y -201.808,Z 1813.780,A 0.000,B 0.000,C 90.000,E1 320.356} C_DIS
LIN {X 0.056,Y -205.754,Z 1813.766,A 0.000,B 0.000,C 90.000,E1 317.919} C_DIS
LIN {X -0.090,Y -210.530,Z 1813.753,A 0.000,B 0.000,C 90.000,E1 315.567} C_DIS
LIN {X 0.101,Y -215.361,Z 1813.742,A 0.000,B 0.000,C 90.000,E1 313.542} C_DIS
LIN {X 0.022,Y -219.873,Z 1813.733,A 0.000,B 0.000,C 90.000,E1 312.000} C_DIS
LIN {X 0.000,Y -225.119,Z 1813.725,A 0.000,B 0.000,C 90.000,E1 310.458} C_DIS
LIN {X 0.073,Y -231.182,Z 1813.716,A 0.000,B 0.000,C 90.000,E1 308.910} C_DIS
LIN {X 0.025,Y -241.501,Z 1813.704,A 0.000,B 0.000,C 90.000,E1 306.664} C_DIS
LIN {X 0.027,Y -253.235,Z 1813.691,A 0.000,B 0.000,C 90.000,E1 304.452} C_DIS
LIN {X 0.038,Y -266.045,Z 1813.679,A 0.000,B 0.000,C 90.000,E1 302.291} C_DIS
LIN {X 0.075,Y -284.827,Z 1813.664,A 0.000,B 0.000,C 90.000,E1 299.489} C_DIS
LIN {X 0.191,Y -297.082,Z 1813.654,A 0.000,B 0.000,C 90.000,E1 297.769} C_DIS
LIN {X 0.170,Y -314.796,Z 1813.642,A 0.000,B 0.000,C 90.000,E1 295.463} C_DIS
LIN {X -0.072,Y -327.515,Z 1813.633,A 0.000,B 0.000,C 90.000,E1 293.898} C_DIS
LIN {X -0.116,Y -340.040,Z 1813.624,A 0.000,B 0.000,C 90.000,E1 292.333} C_DIS
LIN {X -0.107,Y -351.990,Z 1813.615,A 0.000,B 0.000,C 90.000,E1 290.791} C_DIS
LIN {X -0.129,Y -358.697,Z 1813.610,A 0.000,B 0.000,C 90.000,E1 289.885} C_DIS
LIN {X 0.031,Y -364.852,Z 1813.605,A 0.000,B 0.000,C 90.000,E1 288.960} C_DIS
LIN {X 0.135,Y -370.318,Z 1813.600,A 0.000,B 0.000,C 90.000,E1 288.055} C_DIS
LIN {X 0.196,Y -373.505,Z 1813.597,A 0.000,B 0.000,C 90.000,E1 287.457} C_DIS
LIN {X -0.081,Y -376.301,Z 1813.594,A 0.000,B 0.000,C 90.000,E1 286.913} C_DIS
LIN {X 0.020,Y -379.734,Z 1813.589,A 0.000,B 0.000,C 90.000,E1 286.024} C_DIS
LIN {X 0.145,Y -381.609,Z 1813.586,A 0.000,B 0.000,C 90.000,E1 285.426} C_DIS
LIN {X -0.095,Y -383.135,Z 1813.583,A 0.000,B 0.000,C 90.000,E1 284.883} C_DIS
LIN {X -0.052,Y -384.269,Z 1813.579,A 0.000,B 0.000,C 90.000,E1 284.300} C_DIS
LIN {X 0.005,Y -384.951,Z 1813.576,A 0.000,B 0.000,C 90.000,E1 283.716} C_DIS
LIN {X 0.159,Y -385.275,Z 1813.573,A 0.000,B 0.000,C 90.000,E1 283.119} C_DIS
LIN {X -0.147,Y -385.197,Z 1813.570,A 0.000,B 0.000,C 90.000,E1 282.591} C_DIS
LIN {X -0.075,Y -384.669,Z 1813.567,A 0.000,B 0.000,C 90.000,E1 282.007} C_DIS
LIN {X -0.002,Y -383.718,Z 1813.563,A 0.000,B 0.000,C 90.000,E1 281.422} C_DIS
LIN {X 0.067,Y -382.388,Z 1813.560,A 0.000,B 0.000,C 90.000,E1 280.838} C_DIS
LIN {X 0.130,Y -380.689,Z 1813.557,A 0.000,B 0.000,C 90.000,E1 280.254} C_DIS
LIN {X 0.202,Y -377.573,Z 1813.552,A 0.000,B 0.000,C 90.000,E1 279.378} C_DIS
LIN {X 0.184,Y -373.900,Z 1813.547,A 0.000,B 0.000,C 90.000,E1 278.511} C_DIS
LIN {X 0.129,Y -369.668,Z 1813.543,A 0.000,B 0.000,C 90.000,E1 277.644} C_DIS
LIN {X 0.043,Y -364.686,Z 1813.538,A 0.000,B 0.000,C 90.000,E1 276.777} C_DIS
LIN {X -0.091,Y -358.773,Z 1813.533,A 0.000,B 0.000,C 90.000,E1 275.910} C_DIS
LIN {X 0.134,Y -354.217,Z 1813.529,A 0.000,B 0.000,C 90.000,E1 275.277} C_DIS
LIN {X -0.019,Y -348.981,Z 1813.526,A 0.000,B 0.000,C 90.000,E1 274.702} C_DIS
LIN {X -0.119,Y -343.341,Z 1813.523,A 0.000,B 0.000,C 90.000,E1 274.131} C_DIS
LIN {X 0.005,Y -337.393,Z 1813.520,A 0.000,B 0.000,C 90.000,E1 273.555} C_DIS
LIN {X 0.019,Y -331.172,Z 1813.517,A 0.000,B 0.000,C 90.000,E1 273.037} C_DIS
LIN {X -0.065,Y -324.790,Z 1813.514,A 0.000,B 0.000,C 90.000,E1 272.579} C_DIS
LIN {X 0.103,Y -318.205,Z 1813.512,A 0.000,B 0.000,C 90.000,E1 272.121} C_DIS
LIN {X -0.059,Y -311.325,Z 1813.510,A 0.000,B 0.000,C 90.000,E1 271.776} C_DIS
LIN {X 0.061,Y -304.226,Z 1813.508,A 0.000,B 0.000,C 90.000,E1 271.432} C_DIS
LIN {X -0.112,Y -296.702,Z 1813.507,A 0.000,B 0.000,C 90.000,E1 271.203} C_DIS
LIN {X 0.009,Y -289.342,Z 1813.505,A 0.000,B 0.000,C 90.000,E1 270.974} C_DIS
LIN {X -0.121,Y -274.465,Z 1813.504,A 0.000,B 0.000,C 90.000,E1 270.688} C_DIS
LIN {X -0.078,Y -255.800,Z 1813.502,A 0.000,B 0.000,C 90.000,E1 270.344} C_DIS
LIN {X 0.103,Y -246.323,Z 1813.501,A 0.000,B 0.000,C 90.000,E1 270.172} C_DIS
LIN {X -0.026,Y -234.546,Z 1813.501,A 0.000,B 0.000,C 90.000,E1 270.115} C_DIS
LIN {X -0.044,Y -181.573,Z 1813.501,A 0.000,B 0.000,C 90.000,E1 270.115} C_DIS
LIN {X 0.042,Y -180.908,Z 1813.475,A 0.000,B 0.000,C 90.000,E1 265.527} C_DIS
LIN {X -0.081,Y -180.767,Z 1813.471,A 0.000,B 0.000,C 90.000,E1 264.723} C_DIS
LIN {X -0.009,Y -178.861,Z 1813.442,A 0.000,B 0.000,C 90.000,E1 259.634} C_DIS
LIN {X 0.062,Y -175.904,Z 1813.414,A 0.000,B 0.000,C 90.000,E1 254.519} C_DIS
LIN {X 0.000,Y -174.586,Z 1813.405,A 0.000,B 0.000,C 90.000,E1 252.834} C_DIS
LIN {X 0.036,Y -171.568,Z 1813.381,A 0.000,B 0.000,C 90.000,E1 248.539} C_DIS
LIN {X 0.018,Y -167.791,Z 1813.357,A 0.000,B 0.000,C 90.000,E1 244.229} C_DIS
LIN {X 0.032,Y -166.507,Z 1813.347,A 0.000,B 0.000,C 90.000,E1 242.487} C_DIS
LIN {X 0.028,Y -163.216,Z 1813.328,A 0.000,B 0.000,C 90.000,E1 238.997} C_DIS
LIN {X -0.008,Y -161.182,Z 1813.313,A 0.000,B 0.000,C 90.000,E1 236.373} C_DIS
LIN {X -0.009,Y -157.194,Z 1813.289,A 0.000,B 0.000,C 90.000,E1 231.949} C_DIS
LIN {X 0.038,Y -155.923,Z 1813.279,A 0.000,B 0.000,C 90.000,E1 230.150} C_DIS
LIN {X 0.094,Y -152.175,Z 1813.254,A 0.000,B 0.000,C 90.000,E1 225.648} C_DIS
LIN {X 0.003,Y -150.423,Z 1813.239,A 0.000,B 0.000,C 90.000,E1 222.975} C_DIS
LIN {X -0.071,Y -147.150,Z 1813.214,A 0.000,B 0.000,C 90.000,E1 218.463} C_DIS
LIN {X 0.015,Y -145.164,Z 1813.193,A 0.000,B 0.000,C 90.000,E1 214.771} C_DIS
LIN {X -0.068,Y -142.317,Z 1813.162,A 0.000,B 0.000,C 90.000,E1 209.283} C_DIS
LIN {X 0.054,Y -141.707,Z 1813.152,A 0.000,B 0.000,C 90.000,E1 207.385} C_DIS
LIN {X -0.024,Y -139.470,Z 1813.116,A 0.000,B 0.000,C 90.000,E1 200.918} C_DIS
LIN {X 0.030,Y -139.202,Z 1813.106,A 0.000,B 0.000,C 90.000,E1 199.033} C_DIS
LIN {X -0.044,Y -138.328,Z 1813.054,A 0.000,B 0.000,C 90.000,E1 189.726} C_DIS
LIN {X -0.041,Y -139.442,Z 1813.007,A 0.000,B 0.000,C 90.000,E1 181.318} C_DIS
LIN {X 0.038,Y -140.977,Z 1812.976,A 0.000,B 0.000,C 90.000,E1 175.698} C_DIS
LIN {X -0.012,Y -142.732,Z 1812.956,A 0.000,B 0.000,C 90.000,E1 172.008} C_DIS
LIN {X -0.055,Y -145.121,Z 1812.930,A 0.000,B 0.000,C 90.000,E1 167.409} C_DIS
LIN {X -0.060,Y -147.745,Z 1812.910,A 0.000,B 0.000,C 90.000,E1 163.740} C_DIS
LIN {X 0.021,Y -150.411,Z 1812.889,A 0.000,B 0.000,C 90.000,E1 160.061} C_DIS
LIN {X 0.037,Y -153.848,Z 1812.869,A 0.000,B 0.000,C 90.000,E1 156.433} C_DIS
LIN {X -0.046,Y -157.260,Z 1812.849,A 0.000,B 0.000,C 90.000,E1 152.871} C_DIS
